	arrCylinderLink						: ARRAY [0..iMAX_CYLINDER_PAGES-1] OF ARRAY [0..iCYLINDERS_PER_PAGE-1] OF I_UniversalCylinder;				(*  *)
	arrAxisLink							: ARRAY [0..iMAX_AXIS_PAGES-1] OF ARRAY [0..iAXIS_PER_PAGE-1] OF I_UniversalAxis;							(*  *)
	arrInputLink						: ARRAY [0..iMAX_INPUT_PAGES-1] OF ARRAY [0..iINPUTS_PER_PAGE-1] OF I_DigitalInput;							(*  *)
	arrOutputLink						: ARRAY [0..iMAX_OUTPUT_PAGES-1] OF ARRAY [0..iOUTPUTS_PER_PAGE-1] OF I_DigitalOutput;						(*  *)
	arrSafeInputLink					: ARRAY	[0..iMAX_SAFE_INPUT_PAGES-1] OF ARRAY [0..iSAFE_INPUTS_PER_PAGE-1] OF I_DigitalInput;				(*  *)
	arrSafeOutputLink					: ARRAY [0..iMAX_SAFE_OUTPUT_PAGES-1] OF ARRAY [0..iSAFE_OUTPUTS_PER_PAGE-1] OF I_DigitalOutput;			(*  *)
	arrRobotLink						: ARRAY [0..iMAX_ROBOT_PAGES-1] OF ARRAY [0..iROBOTS_PER_PAGE-1] OF I_CR800EtherCAT;						(*  *)
	
	ifUniversalMachineLink				: I_UniversalMachine;	(*  *)
	ifRecipesManager					: I_RecipesManager;		(*  *)
	ifAlarmControler					: I_AlarmControler;		(*  *)
	
	(* --- Alarm page --- *)
	btnClearAll							: BOOL;	(*  *)
	btnExport							: BOOL;	(*  *)
	
	(* --- Recipes page --- *)
	(* Recipe control - buttons *)
	btnCreate							: BOOL;	(* Create recipe button *)
	btnSelect							: BOOL;	(* Select recipe from table button*)
	btnLoad								: BOOL;	(* Load recipe from file button *)
	btnRead								: BOOL;	(* Read recipe to file button *)
	btnReload 							: BOOL;	(* Reload recipes button *)
	btnBackup							: BOOL;	(* Backup recipes to external directory button *)
	btnRestore							: BOOL;	(* Restore recipes from external directory button *)
	btnRemove							: BOOL;	(* Remove recipe from the file *)
	btnReloadExternal					: BOOL;	(* Reload recipes button *)
	btnRecipeNext						: BOOL;	(* Go to next page with recipe parameters *)
	btnRecipePrevious					: BOOL;	(* Go to previous page with recipe parameters *)
	btnHmiClose							: BOOL;
	
	bUpdateVisuElements					: BOOL; (* For function block extending purposes (updating some visualisation elements after loading recipes) *)

	
	(* Recipe control - visibility *)
	bReloadInvisible					: BOOL;	(* Makes reload button invisible *)
	bRecipeNextInvisible				: BOOL;	(* Makes next button invisible *)
	bRecipePreviousInvisible			: BOOL;	(* Makes previous button invisible *)
	bRecipeCreateInvisible				: BOOL;	(* Makes create group box invisible *)
	bRecipeBackupRestoreInvisible		: BOOL;	(* Makes backup and restore group box invisible *)
	bNoRecipeSelected					: BOOL;
	
	(* Recipe control - control disabled *)
	bCreateRecipeDisabled				: BOOL;	(* Disable access to create recipe group box *)
	bBackupRestoreDisabled				: BOOL;	(* Disable access to backup and restore group box *)
	
	(* Recipe control - status *)
	bRecipesManagerError				: REFERENCE TO BOOL;					(* Error occured while executing last command *)
	eRecipesManagerReturns				: REFERENCE TO E_RecipesManagerReturns;	(* Result of last executed command *)
	
	(* Recipe control - parameters for recipes manager *)
	iSelectedRecipe						: INT;												(* Number of selected row in Available Recipes table *)
	sRecipeDefinition					: REFERENCE TO STRING;								(* Name of current recipe definition *)
	sSelectedRecipe						: STRING;											(* Current selected recipe name - changes affter trigger from btnSelect *)
	sNewRecipeName						: STRING;											(* Name for new recipe *)
	sBackupStoragePath					: STRING;											(* Path for backup/restoring of recipes *)
	arrRecipesNames						: REFERENCE TO ARRAY[0..127] OF STRING;				(* Names of all detected recipes *)
	sBackupRestoreRecipeName			: STRING;
		
	(* Recipe control - parameters frame generator *)
	iRecipeParameterIndex 				: USINT := 0;	(*  *)
	iRecipeParameterFrameIndex			: USINT := 0;	(*  *)	
	iRecipeParameterPageIndex			: USINT := 0;	(*  *)
	iSelectedRecipeParameterPageIndex	: USINT := 0;	(*  *)
	
	arrRecipeParameterFrameEmpty 		: ARRAY [0..iMAX_NUMBER_OF_RECIPES-1] OF ARRAY [0..iRECIPE_PARAMETERS_PER_PAGE-1] OF BOOL;							(*  *)
	arrRecipeParameterLink				: ARRAY [0..iMAX_NUMBER_OF_RECIPES-1] OF ARRAY [0..iRECIPE_PARAMETERS_PER_PAGE-1] OF I_RecipeParameter;				(*  *)
	arrRecipeParameterFrameData			: ARRAY [0..iMAX_NUMBER_OF_RECIPES-1] OF ARRAY [0..iRECIPE_PARAMETERS_PER_PAGE-1] OF ST_VisuCtrlRecipeParameter;	(*  *)
	arrRecipeParameterFrameType			: ARRAY [0..iMAX_NUMBER_OF_RECIPES-1] OF ARRAY [0..iRECIPE_PARAMETERS_PER_PAGE-1] OF E_VisuCtrlRecipeParameterType;	(*  *)
	
	(* --- Shell state machines --- *)
	eUniversalMachineCtrlState			: E_VisuCtrUniversalMachineState;		(*  *)
	eRecipesManagerState				: E_VisuCtrlRecipesManagerState;			(* Current state of Recipe Manager *)
	eAlarmCtrlState						: E_VisuCtrlAlarmControlState;			(* Current state of Alarm Controler *)
	
	(* --- Screen selectors --- *)
	eCurrentScreen						: E_VisuCtrlPageState;					(* Main page selector *)
	eLastScreen							: E_VisuCtrlPageState;					(* Last screen before change to auxilary screen *)
	eCurrentNavigation					: E_VisuCtrlNavBarState;				(* Navigation bar selector *)
	
	(* --- HMI buttons flags --- *)
	bStartDisable 						: BOOL;
	bStopDisable						: BOOL	:= TRUE;
	bVisNotInit 						: BOOL	:= TRUE;	
	bVisLogIn							: BOOL;
	bVisLogOut 							: BOOL	:= TRUE;	
	bVisHmiClose						: BOOL;
	bRecipeButtonDisabled				: BOOL;
	bModeSwitchButtonDisabled			: BOOL;
	                        			
	fbHmiClose							: NT_StartProcess;
END_VAR
(*
Version history:

+-------------+------------+----------------+----------+------------------------------------------+
|Date         | Version    | created under  | Author   | Remark                                   |
+=============+============+================+==========+==========================================+
|2022-03      | 1.0.0.0    | V3.1.4024.22   | ADBO     | Function block created                   |
+-------------+------------+----------------+----------+------------------------------------------+

*)

IF bFirstCycle THEN
	bFirstCycle := FALSE;
	(* Assign alarm references *)
	iActiveCriticals	REF= ifAlarmControler.ActiveCritical;
	iActvieErrors 		REF= ifAlarmControler.ActiveError;
	iActiveWarrnings	REF= ifAlarmControler.ActiveWarrning;
	
	(* Assign recipes references *)
	bRecipesManagerError 	REF= ifRecipesManager.Error;
	arrRecipesNames 		REF= ifRecipesManager.RecipesNames;
	eRecipesManagerReturns 	REF= ifRecipesManager.LastResult;
	sRecipeDefinition 		REF= ifRecipesManager.RecipesDefinition;
	
	(* --- Mark unused frames - saves CPU resources --- *)
	(* Cylinder frames *)
	FOR iLoop := 0 TO iMAX_CYLINDER_PAGES-1 DO
		FOR iLoop2 := 0 TO iCYLINDERS_PER_PAGE-1 DO
			IF arrCylinderLink[iLoop][iLoop2] = 0 THEN
				arrCylinderFrameEmpty[iLoop][iLoop2] := TRUE;
			END_IF
		END_FOR
	END_FOR
	
	(* Motor frames *)
	FOR iLoop := 0 TO iMAX_AXIS_PAGES-1 DO
		FOR iLoop2 := 0 TO iAXIS_PER_PAGE-1 DO
			IF arrAxisLink[iLoop][iLoop2] = 0 THEN
				arrAxisFrameEmpty[iLoop][iLoop2] := TRUE;
			END_IF
		END_FOR
	END_FOR
	
	(* Input frames *)
	FOR iLoop := 0 TO iMAX_INPUT_PAGES-1 DO
		FOR iLoop2 := 0 TO iINPUTS_PER_PAGE-1 DO
			IF arrInputLink[iLoop][iLoop2] = 0 THEN
				arrInputFrameEmpty[iLoop][iLoop2] := TRUE;
			END_IF
		END_FOR
	END_FOR
	
	(* Output frames *)
	FOR iLoop := 0 TO iMAX_OUTPUT_PAGES-1 DO
		FOR iLoop2 := 0 TO iOUTPUTS_PER_PAGE-1 DO
			IF arrOutputLink[iLoop][iLoop2] = 0 THEN
				arrOutputFrameEmpty[iLoop][iLoop2] := TRUE;
			END_IF
		END_FOR
	END_FOR
	
	(* Safe input frames *)
	FOR iLoop := 0 TO iMAX_SAFE_INPUT_PAGES-1 DO
		FOR iLoop2 := 0 TO iSAFE_INPUTS_PER_PAGE-1 DO
			IF arrSafeInputLink[iLoop][iLoop2] = 0 THEN
				arrSafeInputFrameEmpty[iLoop][iLoop2] := TRUE;
			END_IF
		END_FOR
	END_FOR
	
	(* Safe output frames *)
	FOR iLoop := 0 TO iMAX_SAFE_OUtPUT_PAGES-1 DO
		FOR iLoop2 := 0 TO iSAFE_OUtPUTS_PER_PAGE-1 DO
			IF arrSafeOutputLink[iLoop][iLoop2] = 0 THEN
				arrSafeOutputFrameEmpty[iLoop][iLoop2] := TRUE;
			END_IF
		END_FOR
	END_FOR
	
	(* Robot frames *)
	FOR iLoop := 0 TO iMAX_ROBOT_PAGES-1 DO
		FOR iLoop2 := 0 TO iROBOTS_PER_PAGE-1 DO
			IF arrRobotLink[iLoop][iLoop2] = 0 THEN
				arrRobotFrameEmpty[iLoop][iLoop2] := TRUE;
			END_IF
		END_FOR
	END_FOR
	
	(* Universal fixture frames *)
	//To-do
	
	(* Tcp-Server frames *)
	// To do
	
	(* Tcp-Client frames*)
	// To do
	
	(* Robot frames *)
	FOR iLoop := 0 TO iMAX_ROBOT_PAGES - 1 DO
		FOR iLoop2 := 0 TO iROBOTS_PER_PAGE - 1 DO
			IF arrRobotLink[iLoop][iLoop2] = 0 THEN
				arrRobotFrameEmpty[iLoop][iLoop2] := TRUE;
			END_IF
		END_FOR
	END_FOR
	
	(* Recipe parameters frames *)
	FOR iLoop := 0 TO iMAX_RECIPES_PAGES-1 DO
		FOR iLoop2 := 0 TO iRECIPE_PARAMETERS_PER_PAGE-1 DO
			IF arrRecipeParameterLink[iLoop][iLoop2] = 0 THEN
				arrRecipeParameterFrameEmpty[iLoop][iLoop2] := TRUE;
			END_IF
		END_FOR
	END_FOR
	
END_IF

(* Get current logged in user *)
IF btnLogIn AND LEN(WSTRING_TO_STRING(VisuUserManagement.VisuElems.CurrentFullUserName)) <> 0 THEN
	sCurrentUser := WSTRING_TO_STRING(VisuUserManagement.VisuElems.CurrentFullUserName);
	btnLogIn := FALSE;
ELSIF btnLogOut THEN
	MEMSET(ADR(sCurrentUser),0,SIZEOF(sCurrentUser));
	btnLogOut := FALSE;
END_IF

(* LogIn and LogOut button status flags *)
IF LEN(sCurrentUser) <> 0 THEN 
	bVisLogIn := TRUE;
	bVisLogOut:= FALSE;
	
ELSE
	bVisLogIn := FALSE;
	bVisLogOut:= TRUE;
	
END_IF

fbHmiClose(
	NETID			:= '',
	PATHSTR			:= 'C:\WINDOWS\system32\taskkill.exe' ,
	DIRNAME			:= '' ,
	COMNDLINE		:= '/t /f /IM Tc3PlcHmi.exe' , 
	START			:= btnHmiClose,
	ERRID			=> );

IF fbHmiClose.BUSY THEN		
	btnHmiClose := FALSE;	
END_IF

(* Get time and date *)
sCurrentDate := FUN_TimestructToDate(fbMachineTime.systemTime);
sCurrentTime := FUN_TimestructToTime(fbMachineTime.systemTime);
sCurrentTime := LEFT(STR := sCurrentTime, SIZE := (LEN(sCurrentTime)-4));

(* Universal switch to Alarms and Recipes page *)
IF btnRecipes THEN
	btnRecipes := FALSE;
	IF eCurrentScreen <> SCREEN_RECIPES AND eCurrentScreen <> SCREEN_ALARMS THEN
		eLastScreen := eCurrentScreen;
	END_IF
	eCurrentScreen := SCREEN_RECIPES;
	
ELSIF btnAlarms THEN
	btnAlarms := FALSE;
	IF eCurrentScreen <> SCREEN_RECIPES AND eCurrentScreen <> SCREEN_ALARMS THEN
		eLastScreen := eCurrentScreen;
	END_IF
	eCurrentScreen := SCREEN_ALARMS;
END_IF

(* Universal change to Abort - Reset mode *)
IF btnAbort THEN
	btnAbort := FALSE;
	eUniversalMachineCtrlState := VISU_CTRL_UNIVERSAL_MACHINE_ABORT;
	eAlarmCtrlState := VISU_CTRL_ALARM_CONTROLER_ABORT;
	eRecipesManagerState := VISU_CTRL_RECIPE_MANAGER_ABORT;
	eRecipesManagerState := VISU_CTRL_RECIPE_MANAGER_INIT;
	eCurrentScreen := SCREEN_ABORTING;
			
ELSIF btnReset THEN
	btnReset := FALSE;
	eUniversalMachineCtrlState := VISU_CTRL_UNIVERSAL_MACHINE_RESET;
END_IF

(* --- Alarm system control via shared interface --- *)
M_AlarmControler();

(* --- Recipes manager control via shared interface --- *)
M_RecipeManager();

(* --- Universal Machine control via shared interface ---*)
M_MachineControler();

(* --- Generic content control state machine --- *)
StateMachine();

PROPERTY Abort : REFERENCE TO BOOL
GET
Abort REF= btnAbort;
END_GET
END_PROPERTY

PROPERTY AutoMode : REFERENCE TO BOOL
GET
AutoMode REF= btnAuto;
END_GET
END_PROPERTY

PROPERTY Back : REFERENCE TO BOOL
GET
Back REF= btnBack;
END_GET
END_PROPERTY

PROPERTY Init : REFERENCE TO BOOL
GET
Init REF= btnInit;
END_GET
END_PROPERTY

METHOD PROTECTED M_AlarmControler
(* --- Active alarms counter --- *)
(*iActiveCriticals := ifAlarmControler.ActiveCritical;
iActvieErrors := ifAlarmControler.ActiveError;
iActiveWarrnings := ifAlarmControler.ActiveWarrning;*)
iActiveAlarms := iActvieErrors + iActiveCriticals;

(* Main alarm control via HMI *)
CASE eAlarmCtrlState OF
	VISU_CTRL_ALARM_CONTROLER_WAIT_FOR_CMD:
		IF btnInit THEN
			eAlarmCtrlState := VISU_CTRL_ALARM_CONTROLER_INIT;
			
		ELSIF btnClearAll THEN
			eAlarmCtrlState := VISU_CTRL_ALARM_CONTROLER_CLEAR_ALL; 
			
		ELSIF btnExport THEN
			eAlarmCtrlState := VISU_CTRL_ALARM_CONTTOLER_EXPORT;
			
		END_IF
		
	VISU_CTRL_ALARM_CONTROLER_INIT:
		ifAlarmControler.MR_Init();
		
		IF ifAlarmControler.Active THEN
			eAlarmCtrlState := VISU_CTRL_ALARM_CONTROLER_WAIT_FOR_CMD;
		END_IF
		
	VISU_CTRL_ALARM_CONTROLER_CLEAR_ALL:
		ifAlarmControler.MR_ClearAll(bResetConfirmation := TRUE);
		
		IF NOT ifAlarmControler.Busy THEN
			eAlarmCtrlState := VISU_CTRL_ALARM_CONTROLER_WAIT_FOR_CMD;
		END_IF
	
	VISU_CTRL_ALARM_CONTTOLER_EXPORT:
		ifAlarmControler.MR_Export();
		
		IF NOT ifAlarmControler.Busy THEN
			eAlarmCtrlState := VISU_CTRL_ALARM_CONTROLER_WAIT_FOR_CMD;
		END_IF
		
	VISU_CTRL_ALARM_CONTROLER_ABORT:
		ifAlarmControler.MR_Abort();
		
		IF NOT ifAlarmControler.Active THEN
			eAlarmCtrlState := VISU_CTRL_ALARM_CONTROLER_WAIT_FOR_CMD;
		END_IF
		
END_CASE
END_METHOD

METHOD M_MachineControler : BOOL
(* Main machine control via HMI *)
IF NOT ifUniversalMachineLink.Running THEN
	bStartDisable := FALSE;
	bStopDisable := TRUE;
ELSE
	bStartDisable := TRUE;
	bStopDisable := FALSE;
END_IF

CASE eUniversalMachineCtrlState OF
	VISU_CTRL_UNIVERSAL_MACHINE_WAIT_FOR_CMD:
		IF btnInit THEN
			eUniversalMachineCtrlState := VISU_CTRL_UNIVERSAL_MACHINE_INIT;
			
		ELSIF btnStart THEN
			eUniversalMachineCtrlState := VISU_CTRL_UNIVERSAL_MACHINE_START_AUTO;
			
		ELSIF btnStop THEN
			eUniversalMachineCtrlState := VISU_CTRL_UNIVERSAL_MACHINE_STOP_AUTO;
			
		ELSIF btnManual THEN
			eUniversalMachineCtrlState := VISU_CTRL_UNIVERSAL_MACHINE_SWITCH_TO_MANUAL;
			
		ELSIF btnAuto THEN
			eUniversalMachineCtrlState := VISU_CTRL_UNIVERSAL_MACHINE_SWITCH_TO_AUTO;
			
		ELSIF btnAbort THEN
			eUniversalMachineCtrlState := VISU_CTRL_UNIVERSAL_MACHINE_ABORT;
			
		ELSIF btnReset THEN
			eUniversalMachineCtrlState := VISU_CTRL_UNIVERSAL_MACHINE_RESET;			
		END_IF
	
	VISU_CTRL_UNIVERSAL_MACHINE_INIT:
		ifUniversalMachineLink.MR_Init();
		
		IF ifUniversalMachineLink.Active THEN
			bVisNotInit := FALSE;
			bVisHmiClose:= TRUE;
						
			eUniversalMachineCtrlState := VISU_CTRL_UNIVERSAL_MACHINE_WAIT_FOR_CMD;
		END_IF
	
	VISU_CTRL_UNIVERSAL_MACHINE_RESET:
		ifUniversalMachineLink.MR_Reset();
		
		IF NOT ifUniversalMachineLink.Error THEN
			eUniversalMachineCtrlState := VISU_CTRL_UNIVERSAL_MACHINE_WAIT_FOR_CMD;
		END_IF
	
	VISU_CTRL_UNIVERSAL_MACHINE_START_AUTO:
		ifUniversalMachineLink.MR_Start();
		
		IF ifUniversalMachineLink.Running THEN
			eUniversalMachineCtrlState := VISU_CTRL_UNIVERSAL_MACHINE_WAIT_FOR_CMD;
		END_IF
	
	VISU_CTRL_UNIVERSAL_MACHINE_STOP_AUTO:
		ifUniversalMachineLink.MR_Stop();
		
		IF NOT ifUniversalMachineLink.Running THEN
			eUniversalMachineCtrlState := VISU_CTRL_UNIVERSAL_MACHINE_WAIT_FOR_CMD;
		END_IF
		
	VISU_CTRL_UNIVERSAL_MACHINE_SWITCH_TO_MANUAL:
		ifUniversalMachineLink.MR_SwitchToManual();
		
		IF ifUniversalMachineLink.State = MACHINE_STATE_MANUAL THEN
			eUniversalMachineCtrlState := VISU_CTRL_UNIVERSAL_MACHINE_WAIT_FOR_CMD;
		END_IF
	
	VISU_CTRL_UNIVERSAL_MACHINE_SWITCH_TO_AUTO:
		ifUniversalMachineLink.MR_SwitchToAuto();
		
		IF ifUniversalMachineLink.State = MACHINE_STATE_AUTO THEN
			eUniversalMachineCtrlState := VISU_CTRL_UNIVERSAL_MACHINE_WAIT_FOR_CMD;
		END_IF
	
	VISU_CTRL_UNIVERSAL_MACHINE_ABORT:
		ifUniversalMachineLink.MR_Abort();
		
		IF NOT ifUniversalMachineLink.Active THEN
			bVisNotInit := TRUE;
			bVisHmiClose:= FALSE;
			
			eUniversalMachineCtrlState := VISU_CTRL_UNIVERSAL_MACHINE_WAIT_FOR_CMD;
		END_IF
		
END_CASE
END_METHOD

METHOD PROTECTED M_RecipeManager
bRecipesManagerError 	:= ifRecipesManager.Error;
arrRecipesNames 		:= ifRecipesManager.RecipesNames;
eRecipesManagerReturns 	:= ifRecipesManager.LastResult;
sRecipeDefinition 		:= ifRecipesManager.RecipesDefinition;

IF bStartDisable OR bVisNotInit THEN
	bRecipeButtonDisabled := TRUE;
ELSE
	bRecipeButtonDisabled := FALSE;
END_IF

(* Previous page button visiblity control *)
IF iSelectedRecipeParameterPageIndex = 0 THEN
	bRecipePreviousInvisible := TRUE;
ELSE
	bRecipePreviousInvisible := FALSE;
END_IF

IF sSelectedRecipe = '' THEN
	bNoRecipeSelected := TRUE;

ELSE 
	bNoRecipeSelected := FALSE;

END_IF

(* Next page button visibility control *)
IF btnRecipeNext THEN
	btnRecipeNext := FALSE;
	iSelectedRecipeParameterPageIndex := iSelectedRecipeParameterPageIndex + 1;
	
ELSIF btnRecipePrevious THEN
	btnRecipePrevious := FALSE;
	iSelectedRecipeParameterPageIndex := iSelectedRecipeParameterPageIndex - 1;
END_IF

(* Selecting new recipe from table *)
IF btnSelect THEN
	btnSelect := FALSE;
	sSelectedRecipe	:= arrRecipesNames[iSelectedRecipe];
	eRecipesManagerState := VISU_CTRL_RECIPE_MANAGER_RELOAD;
END_IF

(* Main recipe manager control via HMI *)
CASE eRecipesManagerState OF
	VISU_CTRL_RECIPE_MANAGER_WAIT_FOR_CMD:
		IF btnInit THEN
			eRecipesManagerState := VISU_CTRL_RECIPE_MANAGER_INIT;
			
		ELSIF btnCreate THEN
			btnCreate := FALSE;
			eRecipesManagerState := VISU_CTRL_RECIPE_MANAGER_CREATE;
			
		ELSIF btnLoad THEN
			btnLoad := FALSE;
			eRecipesManagerState := VISU_CTRL_RECIPE_MANAGER_LOAD;
			
		ELSIF btnRead THEN
			btnRead := FALSE;
			eRecipesManagerState := VISU_CTRL_RECIPE_MANAGER_READ;
			
		ELSIF btnReload THEN
			btnReload := FALSE;
			eRecipesManagerState := VISU_CTRL_RECIPE_MANAGER_RELOAD;	
						
		ELSIF btnReloadExternal THEN
			btnReloadExternal := FALSE;
			eRecipesManagerState := VISU_CTRL_RECIPE_MANAGER_RELOAD_EXT;
			
		ELSIF btnBackup THEN
			btnBackup := FALSE;
			eRecipesManagerState := VISU_CTRL_RECIPE_MANAGER_BACKUP;
			
		ELSIF btnRestore THEN
			btnRestore := FALSE;
			eRecipesManagerState := VISU_CTRL_RECIPE_MANAGER_RESTORE;
			
		ELSIF btnRemove THEN
			btnRemove := FALSE;
			eRecipesManagerState := VISU_CTRL_RECIPE_MANAGER_REMOVE;
						
		END_IF
		
	VISU_CTRL_RECIPE_MANAGER_INIT:
		ifRecipesManager.MR_Init();
		
		IF ifRecipesManager.Active THEN
			eRecipesManagerState := VISU_CTRL_RECIPE_MANAGER_WAIT_FOR_CMD;
		END_IF
	
	VISU_CTRL_RECIPE_MANAGER_CREATE:
		ifRecipesManager.MR_Create( sRecipesDefinition	:= sRecipeDefinition,
									sRecipeName			:= sNewRecipeName);
									
		IF NOT ifRecipesManager.Busy THEN
			eRecipesManagerState := VISU_CTRL_RECIPE_MANAGER_WAIT_FOR_CMD;
		END_IF
	
	VISU_CTRL_RECIPE_MANAGER_LOAD:
		ifRecipesManager.MR_LoadAndWritte( 	sRecipesDefinition	:= sRecipeDefinition,
											sRecipeName			:= sSelectedRecipe);
									
		IF NOT ifRecipesManager.Busy THEN
			IF NOT ifRecipesManager.Error THEN
				sCurrentRecipe := sSelectedRecipe; 
			END_IF
			
			bUpdateVisuElements := TRUE;
			eRecipesManagerState := VISU_CTRL_RECIPE_MANAGER_WAIT_FOR_CMD;
		END_IF
	
	VISU_CTRL_RECIPE_MANAGER_READ:
		ifRecipesManager.MR_ReadAndSave(	sRecipesDefinition	:= sRecipeDefinition,
											sRecipeName			:= sSelectedRecipe);
									
		IF NOT ifRecipesManager.Busy THEN
			eRecipesManagerState := VISU_CTRL_RECIPE_MANAGER_WAIT_FOR_CMD;
		END_IF
	
	VISU_CTRL_RECIPE_MANAGER_RELOAD:
		ifRecipesManager.MR_Reload( sRecipesDefinition := sRecipeDefinition,
									sRecipeName := sSelectedRecipe);
									
		IF NOT ifRecipesManager.Busy THEN
			eRecipesManagerState := VISU_CTRL_RECIPE_MANAGER_WAIT_FOR_CMD;
		END_IF
		
	VISU_CTRL_RECIPE_MANAGER_RELOAD_EXT:
		ifRecipesManager.MR_ReloadExternal( sRecipesDefinition := sRecipeDefinition,
											sRecipeName := sBackupRestoreRecipeName,
											sBackupStoragePath := sBackupStoragePath);
									
		IF NOT ifRecipesManager.Busy THEN
			eRecipesManagerState := VISU_CTRL_RECIPE_MANAGER_WAIT_FOR_CMD;
		END_IF	
	
	VISU_CTRL_RECIPE_MANAGER_BACKUP:
		ifRecipesManager.MR_Backup(sRecipesDefinition := sRecipeDefinition,
									sRecipeName := sBackupRestoreRecipeName,
									sBackupStoragePath := sBackupStoragePath);
									
		IF NOT ifRecipesManager.Busy THEN
			eRecipesManagerState := VISU_CTRL_RECIPE_MANAGER_WAIT_FOR_CMD;
		END_IF
		
	VISU_CTRL_RECIPE_MANAGER_RESTORE:
		ifRecipesManager.MR_Restore(sRecipesDefinition := sRecipeDefinition,
									sRecipeName := sBackupRestoreRecipeName,
									sBackupStoragePath := sBackupStoragePath);
									
		IF NOT ifRecipesManager.Busy THEN
			IF NOT ifRecipesManager.Error THEN
				sCurrentRecipe := sSelectedRecipe; 
			END_IF
			
			bUpdateVisuElements := TRUE;
			eRecipesManagerState := VISU_CTRL_RECIPE_MANAGER_WAIT_FOR_CMD;
		END_IF
		
	VISU_CTRL_RECIPE_MANAGER_REMOVE:
		ifRecipesManager.MR_Remove( sRecipesDefinition := sRecipeDefinition,
									sRecipeName := sSelectedRecipe);
		
		IF NOT ifRecipesManager.Busy THEN
			eRecipesManagerState := VISU_CTRL_RECIPE_MANAGER_WAIT_FOR_CMD;
		END_IF
	
	VISU_CTRL_RECIPE_MANAGER_ABORT:
		ifRecipesManager.MR_Abort();
		
		IF NOT ifRecipesManager.Active THEN
			eRecipesManagerState := VISU_CTRL_RECIPE_MANAGER_WAIT_FOR_CMD;
		END_IF
	
END_CASE
END_METHOD

PROPERTY ManualMode : REFERENCE TO BOOL
GET
ManualMode REF= btnManual;
END_GET
END_PROPERTY

METHOD MR_AppendAlarmControler : BOOL
VAR_INPUT
	ifAlarmControler : I_AlarmControler;
END_VAR
THIS^.ifAlarmControler := ifAlarmControler;
MR_AppendAlarmControler := TRUE;
END_METHOD

METHOD MR_AppendAxis : BOOL
VAR_INPUT
	ifMotor 	: I_UniversalAxis;
	eMotorType	: E_VisuCtrlAxisImgType;
END_VAR
IF iAxisIndex < iMAX_AXIS_FRAMES THEN
	arrAxisLink[iAxisPageIndex][iAxisFrameIndex] := ifMotor;
	arrAxisFrameEmpty[iAxisPageIndex][iAxisFrameIndex] := FALSE;
	arrAxisFrame[iAxisPageIndex][iAxisFrameIndex].sAxisImage := TO_STRING(eMotorType);
	
	IF iAxisFrameIndex = iAXIS_PER_PAGE - 1 THEN
		iAxisPageIndex := iAxisPageIndex + 1;
		iAxisFrameIndex := 0;
	ELSE
		iAxisFrameIndex := iAxisFrameIndex + 1;
	END_IF	

	iAxisIndex := iAxisIndex + 1;
	MR_AppendAxis := TRUE;
ELSE
	MR_AppendAxis := FALSE;
END_IF
END_METHOD

METHOD MR_AppendCylinder : BOOL
VAR_INPUT
	ifCylinder			: I_UniversalCylinder;
	eCylinderType		: E_VisuCtrlCylinderImgType;
	sActiveDescription	: STRING;
	sHomeDescription	: STRING;
END_VAR
IF iCylinderIndex < iMAX_CYLINDER_FRAMES THEN
	arrCylinderLink[iCylinderPageIndex][iCylinderFrameIndex] := ifCylinder;
	arrCylinderFrameEmpty[iCylinderPageIndex][iCylinderFrameIndex] := FALSE;
	
	arrCylinderFrame[iCylinderPageIndex][iCylinderFrameIndex].sCylinderImage := TO_STRING(eCylinderType);
	arrCylinderFrame[iCylinderPageIndex][iCylinderFrameIndex].sActiveDescription := sActiveDescription;
	arrCylinderFrame[iCylinderPageIndex][iCylinderFrameIndex].sHomeDescription := sHomeDescription;
	
	IF iCylinderFrameIndex = iCYLINDERS_PER_PAGE - 1 THEN
		iCylinderPageIndex := iCylinderPageIndex + 1;
		iCylinderFrameIndex := 0;
	ELSE
		iCylinderFrameIndex := iCylinderFrameIndex + 1;
	END_IF	

	iCylinderIndex := iCylinderIndex + 1;
	MR_AppendCylinder := TRUE;
ELSE
	MR_AppendCylinder := FALSE;
END_IF
END_METHOD

METHOD MR_AppendInput : BOOL
VAR_INPUT
	ifDigitalInput : I_DigitalInput;
END_VAR
IF iInputIndex < iMAX_INPUT_FRAMES THEN
	arrInputLink[iInputPageIndex][iInputFrameIndex] := ifDigitalInput;
	arrInputFrameEmpty[iInputPageIndex][iInputFrameIndex] := FALSE;
	
	IF iInputFrameIndex = iINPUTS_PER_PAGE - 1 THEN
		iInputPageIndex := iInputPageIndex + 1;
		iInputFrameIndex := 0;
	ELSE
		iInputFrameIndex := iInputFrameIndex + 1;
	END_IF	
	
	iInputIndex := iInputIndex + 1;
	MR_AppendInput := TRUE;
ELSE
	MR_AppendInput := FALSE;
END_IF
END_METHOD

METHOD MR_AppendOutput : BOOL
VAR_INPUT
	ifDigitalOutput : I_DigitalOutput;
END_VAR
IF iOutputIndex < iMAX_OUTPUT_FRAMES THEN
	arrOutputLink[iOutputPageIndex][iOutputFrameIndex] := ifDigitalOutput;
	arrOutputFrameEmpty[iOutputPageIndex][iOutputFrameIndex] := FALSE;
	
	IF iOutputFrameIndex = iOUTPUTS_PER_PAGE - 1 THEN
		iOutputPageIndex := iOutputPageIndex + 1;
		iOutputFrameIndex := 0;
	ELSE
		iOutputFrameIndex := iOutputFrameIndex + 1;
	END_IF	

	iOutputIndex := iOutputIndex + 1;
	MR_AppendOutput := TRUE;
ELSE
	MR_AppendOutput := FALSE;
END_IF
END_METHOD

METHOD MR_AppendRecipeParameter : BOOL
VAR_INPUT
	ifRecipeParameter : I_RecipeParameter;
END_VAR
IF iRecipeParameterIndex < iMAX_NUMBER_OF_RECIPES THEN
	arrRecipeParameterLink[iRecipeParameterPageIndex][iRecipeParameterFrameIndex] 		:= ifRecipeParameter;
	arrRecipeParameterFrameEmpty[iRecipeParameterPageIndex][iRecipeParameterFrameIndex] := FALSE;
	arrRecipeParameterFrameType[iRecipeParameterPageIndex][iRecipeParameterFrameIndex]	:= ifRecipeParameter.DataType;
	
	arrRecipeParameterFrameData[iRecipeParameterPageIndex][iRecipeParameterFrameIndex].bValue 		REF= arrRecipeParameterLink[iRecipeParameterPageIndex][iRecipeParameterFrameIndex].BitValue;
	arrRecipeParameterFrameData[iRecipeParameterPageIndex][iRecipeParameterFrameIndex].iValue 		REF= arrRecipeParameterLink[iRecipeParameterPageIndex][iRecipeParameterFrameIndex].IntValue;
	arrRecipeParameterFrameData[iRecipeParameterPageIndex][iRecipeParameterFrameIndex].rValue 		REF= arrRecipeParameterLink[iRecipeParameterPageIndex][iRecipeParameterFrameIndex].RealValue;
	arrRecipeParameterFrameData[iRecipeParameterPageIndex][iRecipeParameterFrameIndex].sValue 		REF= arrRecipeParameterLink[iRecipeParameterPageIndex][iRecipeParameterFrameIndex].StringValue;
	arrRecipeParameterFrameData[iRecipeParameterPageIndex][iRecipeParameterFrameIndex].sName 		REF= arrRecipeParameterLink[iRecipeParameterPageIndex][iRecipeParameterFrameIndex].Name;
	arrRecipeParameterFrameData[iRecipeParameterPageIndex][iRecipeParameterFrameIndex].sFileValue 	REF= arrRecipeParameterLink[iRecipeParameterPageIndex][iRecipeParameterFrameIndex].FileValue;
	
	IF iRecipeParameterFrameIndex = iRECIPE_PARAMETERS_PER_PAGE - 1 THEN
		iRecipeParameterPageIndex := iRecipeParameterPageIndex + 1;
		iRecipeParameterFrameIndex := 0;
	ELSE
		iRecipeParameterFrameIndex := iRecipeParameterFrameIndex + 1;
	END_IF	
	
	iRecipeParameterIndex := iRecipeParameterIndex + 1;
	MR_AppendRecipeParameter := FALSE;
ELSE
	MR_AppendRecipeParameter := FALSE;
END_IF
END_METHOD

METHOD MR_AppendRecipesManager : BOOL
VAR_INPUT
	ifRecipesManager : I_RecipesManager;
END_VAR
THIS^.ifRecipesManager := ifRecipesManager;
MR_AppendRecipesManager := TRUE;
END_METHOD

METHOD MR_AppendRobot : BOOL
VAR_INPUT
	ifRobot				: I_CR800EtherCAT;
	eRobotType			: E_VisuCtrlRobotImgType;
//	sErrorDescription	: STRING;
END_VAR
IF iRobotIndex < iMAX_ROBOT_FRAMES THEN
	arrRobotLink[iRobotPageIndex][iRobotFrameIndex] := ifRobot;
	arrRobotFrameEmpty[iRobotPageIndex][iRobotFrameIndex] := FALSE;
	arrRobotFrame[iRobotPageIndex][iRobotFrameIndex].sRobotImage := TO_STRING(eRobotType);
	
	IF iRobotFrameIndex = iROBOTS_PER_PAGE - 1 THEN
		iRobotPageIndex := iRobotPageIndex + 1;
		iRobotFrameIndex := 0;
	ELSE
		iRobotFrameIndex := iRobotFrameIndex + 1;
	END_IF	

	iRobotIndex := iRobotIndex + 1;
	MR_AppendRobot := TRUE;
ELSE
	MR_AppendRobot := FALSE;
END_IF
END_METHOD

METHOD MR_AppendSafeInput : BOOL
VAR_INPUT
	ifSafeInput : I_DigitalInput;
END_VAR
IF iSafeInputIndex < iMAX_SAFE_INPUT_FRAMES THEN
	arrSafeInputLink[iSafeInputPageIndex][iSafeInputFrameIndex] := ifSafeInput;
	arrSafeInputFrameEmpty[iSafeInputPageIndex][iSafeInputFrameIndex] := FALSE;
	
	IF iSafeInputFrameIndex = iSAFE_INPUTS_PER_PAGE - 1 THEN
		iSafeInputPageIndex := iSafeInputPageIndex + 1;
		iSafeInputFrameIndex := 0;
	ELSE
		iSafeInputFrameIndex := iSafeInputFrameIndex + 1;
	END_IF	
	
	iSafeInputIndex := iSafeInputIndex + 1;
	MR_AppendSafeInput := TRUE;
ELSE
	MR_AppendSafeInput := FALSE;
END_IF
END_METHOD

METHOD MR_AppendSafeOutput : BOOL
VAR_INPUT
	ifSafeOutput : I_DigitalOutput;
END_VAR
IF iSafeOutputIndex < iMAX_SAFE_OUTPUT_FRAMES THEN
	arrSafeOutputLink[iSafeOutputPageIndex][iSafeOutputFrameIndex] := ifSafeOutput;
	arrSafeOutputFrameEmpty[iSafeOutputPageIndex][iSafeOutputFrameIndex] := FALSE;
	
	IF iSafeOutputFrameIndex = iSAFE_OUTPUTS_PER_PAGE - 1 THEN
		iSafeOutputPageIndex := iSafeOutputPageIndex + 1;
		iSafeOutputFrameIndex := 0;
	ELSE
		iSafeOutputFrameIndex := iSafeOutputFrameIndex + 1;
	END_IF		

	iSafeOutputIndex := iSafeOutputIndex + 1;
	MR_AppendSafeOutput := TRUE;
ELSE
	MR_AppendSafeOutput := FALSE;
END_IF
END_METHOD

METHOD MR_AppendUniversalMachine : BOOL
VAR_INPUT
	ifMachine : I_UniversalMachine;
END_VAR
THIS^.ifUniversalMachineLink := ifMachine;
MR_AppendUniversalMachine := TRUE;
END_METHOD

METHOD MR_FirstCycle : BOOL
VAR_INPUT
	sMachineName : STRING;
	sSoftwareVersion : STRING;
END_VAR
THIS^.sMachineName := sMachineName;
THIS^.sSoftwareVersion := sSoftwareVersion;
END_METHOD

METHOD PROTECTED MS_Aborting
VAR_INPUT
END_VAR
eCurrentNavigation := NAVIGATION_EMPTY;

IF ifUniversalMachineLink.State = MACHINE_STATE_UNINITIALIZED THEN
	eCurrentScreen := SCREEN_UNINITIALIZED;
	
ELSIF ifUniversalMachineLink.State = MACHINE_STATE_EMERGENCY THEN
	eCurrentScreen := SCREEN_EMERGENCY;
	
END_IF
END_METHOD

METHOD PROTECTED MS_Alarms
VAR_INPUT
END_VAR
eCurrentNavigation := NAVIGATION_UTILITIES;

IF btnBack THEN
	btnBack := FALSE;
	eCurrentScreen := eLastScreen;
END_IF
END_METHOD

METHOD PROTECTED MS_Auto
VAR_INPUT
END_VAR
eCurrentNavigation := NAVIGATION_AUTO;

IF ifUniversalMachineLink.State = MACHINE_STATE_ABORTING THEN
	eCurrentScreen := SCREEN_ABORTING;	

ELSIF ifUniversalMachineLink.State = MACHINE_STATE_AUTO_TO_MANUAL THEN
	eCurrentScreen := SCREEN_MODE_CHANGE;
	
	IF iOutputIndex > 0 THEN
		FOR iLoop := 0 TO iOUTPUTS_PER_PAGE-1 DO
			IF arrOutputFrameEmpty[iSelectedOutputPageIndex][iLoop] = FALSE THEN
				arrOutputFrame[iSelectedOutputPageIndex][iLoop].btnOut := arrOutputLink[iSelectedOutputPageIndex][iLoop].Out;
				
				IF arrOutputFrameEmpty[iSelectedOutputPageIndex][iLoop +1 ] = TRUE THEN
					EXIT;
					
				END_IF
			END_IF
		END_FOR
	END_IF
ELSIF ifUniversalMachineLink.State = MACHINE_STATE_EMERGENCY THEN
	eCurrentScreen := SCREEN_EMERGENCY;
	
END_IF
END_METHOD

METHOD PROTECTED ABSTRACT MS_Emergency
END_METHOD

METHOD PROTECTED MS_Initializing
VAR_INPUT
END_VAR
eCurrentNavigation := NAVIGATION_INITIALIZING;

IF ifUniversalMachineLink.State = MACHINE_STATE_UNINITIALIZED THEN
	eCurrentScreen := SCREEN_UNINITIALIZED;
			
ELSIF ifUniversalMachineLink.State = MACHINE_STATE_READY_INITIALIZED THEN
	eCurrentScreen := SCREEN_READY_INITIALIZED;
	
ELSIF ifUniversalMachineLink.State = MACHINE_STATE_AUTO THEN
	eCurrentScreen := SCREEN_AUTO;
	
ELSIF ifUniversalMachineLink.State = MACHINE_STATE_EMERGENCY THEN
	eCurrentScreen := SCREEN_EMERGENCY;
			
END_IF
END_METHOD

METHOD PROTECTED MS_Manual
VAR_INPUT
END_VAR
eCurrentNavigation := NAVIGATION_MANUAL;

IF ifUniversalMachineLink.State = MACHINE_STATE_UNINITIALIZED THEN
	eCurrentScreen := SCREEN_UNINITIALIZED;	
	
ELSIF ifUniversalMachineLink.State = MACHINE_STATE_MANUAL_TO_AUTO THEN
	eCurrentScreen := SCREEN_MODE_CHANGE;
	
ELSIF ifUniversalMachineLink.State = MACHINE_STATE_EMERGENCY THEN
	eCurrentScreen := SCREEN_EMERGENCY;
	
END_IF

IF btnManualCylinder THEN
	eCurrentScreen := SCREEN_MANUAL_CYLINDERS;

ELSIF btnManualAxis THEN
	eCurrentScreen := SCREEN_MANUAL_MOTORS;
	
ELSIF btnManualInputs THEN
	eCurrentScreen := SCREEN_MANUAL_INPUTS;
	
ELSIF btnManualOutputs THEN
	eCurrentScreen := SCREEN_MANUAL_OUTPUTS;
	
//ELSIF btnManualSafety THEN
//	eCurrentScreen := SCREEN_MANUAL_SAFETY;

ELSIF btnManualRobots THEN
	eCurrentScreen := SCREEN_MANUAL_ROBOTS;

ELSIF btnManualOthers THEN
	eCurrentScreen := SCREEN_MANUAL_OTHERS;
	
END_IF
END_METHOD

METHOD PROTECTED MS_ManualAxis
VAR_INPUT
END_VAR
(*Set current screen *)
eCurrentScreen := SCREEN_MANUAL_MOTORS;

(* Run common part of manual pages handling *)
MS_Manual();

IF arrAxisFrameEmpty[iAxisPageIndex][0] THEN
    iAxisPageIndex := iAxisPageIndex - 1;
END_IF

bNextInvisible := iSelectedAxisPageIndex = iAxisPageIndex;
bPreviousInvisible := iSelectedAxisPageIndex = 0;

(* Frames control *)
IF btnPrevious THEN
	btnPrevious := FALSE;
	iSelectedAxisPageIndex := iSelectedAxisPageIndex - 1;
ELSIF btnNext THEN
	btnNext := FALSE;
	iSelectedAxisPageIndex := iSelectedAxisPageIndex + 1;
END_IF

IF iAxisIndex > 0 THEN
	FOR iLoop := 0 TO iAXIS_PER_PAGE-1 DO
		IF arrAxisFrameEmpty[iSelectedAxisPageIndex][iLoop] = FALSE THEN
			(* Assign object status to frame*)
			arrAxisFrame[iSelectedAxisPageIndex][iLoop].bActive := arrAxisLink[iSelectedAxisPageIndex][iLoop].Active;
			arrAxisFrame[iSelectedAxisPageIndex][iLoop].bHomed := arrAxisLink[iSelectedAxisPageIndex][iLoop].IsHomed;
			arrAxisFrame[iSelectedAxisPageIndex][iLoop].bInPosition := arrAxisLink[iSelectedAxisPageIndex][iLoop].InPosition;
			arrAxisFrame[iSelectedAxisPageIndex][iLoop].bHalted := arrAxisLink[iSelectedAxisPageIndex][iLoop].Halted;
			arrAxisFrame[iSelectedAxisPageIndex][iLoop].bError := arrAxisLink[iSelectedAxisPageIndex][iLoop].Error;
			arrAxisFrame[iSelectedAxisPageIndex][iLoop].iErrorID := arrAxisLink[iSelectedAxisPageIndex][iLoop].ErrorID;
			arrAxisFrame[iSelectedAxisPageIndex][iLoop].eAxisState := arrAxisLink[iSelectedAxisPageIndex][iLoop].State;
			arrAxisFrame[iSelectedAxisPageIndex][iLoop].lrActualPosition := arrAxisLink[iSelectedAxisPageIndex][iLoop].ActualPosition;
			arrAxisFrame[iSelectedAxisPageIndex][iLoop].lrActualVelocity := arrAxisLink[iSelectedAxisPageIndex][iLoop].ActualVelocity;
			arrAxisFrame[iSelectedAxisPageIndex][iLoop].lrSetPosition := arrAxisLink[iSelectedAxisPageIndex][iLoop].SetpointPosition;
			arrAxisFrame[iSelectedAxisPageIndex][iLoop].lrSetVelocity := arrAxisLink[iSelectedAxisPageIndex][iLoop].SetpointVelocity;
			arrAxisFrame[iSelectedAxisPageIndex][iLoop].lrLagError := arrAxisLink[iSelectedAxisPageIndex][iLoop].LagError;
			arrAxisFrame[iSelectedAxisPageIndex][iLoop].sName := arrAxisLink[iSelectedAxisPageIndex][iLoop].Name;
			arrAxisFrame[iSelectedAxisPageIndex][iLoop].sUnit := arrAxisLink[iSelectedAxisPageIndex][iLoop].Unit;
			
			(* Assign parameters from frame to object *)
			arrAxisLink[iSelectedAxisPageIndex][iLoop].Override := arrAxisFrame[iSelectedAxisPageIndex][iLoop].lrOverride;
			arrAxisLink[iSelectedAxisPageIndex][iLoop].JogPosition := arrAxisFrame[iSelectedAxisPageIndex][iLoop].lrJogDistance;
			arrAxisLink[iSelectedAxisPageIndex][iLoop].JogVelocity := arrAxisFrame[iSelectedAxisPageIndex][iLoop].lrJogVelocity;
			arrAxisLink[iSelectedAxisPageIndex][iLoop].JogAcceleration := arrAxisFrame[iSelectedAxisPageIndex][iLoop].lrJogAcceleration;
			arrAxisLink[iSelectedAxisPageIndex][iLoop].JogDeceleration := arrAxisFrame[iSelectedAxisPageIndex][iLoop].lrJogDeceleartion;
			
			(* Bound jog mode frame selector to axis object jog mode *)
			CASE arrAxisFrame[iSelectedAxisPageIndex][iLoop].eJogMode OF
				VISU_AXIS_JOG_MODE_STANDARD_SLOW:
					arrAxisLink[iSelectedAxisPageIndex][iLoop].JogMode := E_JogMode.MC_JOGMODE_STANDARD_SLOW;
					
				VISU_AXIS_JOG_MODE_STANDARD_FAST:
					arrAxisLink[iSelectedAxisPageIndex][iLoop].JogMode := E_JogMode.MC_JOGMODE_STANDARD_FAST;
					
				VISU_AXIS_JOG_MODE_CONTINOUS:
					arrAxisLink[iSelectedAxisPageIndex][iLoop].JogMode := E_JogMode.MC_JOGMODE_CONTINOUS;
					
				VISU_AXIS_JOG_MODE_INCHING:
					arrAxisLink[iSelectedAxisPageIndex][iLoop].JogMode := E_JogMode.MC_JOGMODE_INCHING;
					
				VISU_AXIS_JOG_MODE_INCHING_MODULO:
					arrAxisLink[iSelectedAxisPageIndex][iLoop].JogMode := E_JogMode.MC_JOGMODE_INCHING_MODULO;
					
			END_CASE
			
			(* Manual object control via requests *)
			IF arrAxisFrame[iSelectedAxisPageIndex][iLoop].btnReset THEN
				arrAxisFrame[iSelectedAxisPageIndex][iLoop].btnReset := FALSE;
				arrAxisState[iSelectedAxisPageIndex][iLoop] := VISU_CTRL_AXIS_RESET;
				
			ELSIF arrAxisFrame[iSelectedAxisPageIndex][iLoop].btnHalt THEN
				arrAxisFrame[iSelectedAxisPageIndex][iLoop].btnHalt := FALSE;
				arrAxisState[iSelectedAxisPageIndex][iLoop] := VISU_CTRL_AXIS_HALT;
				
			END_IF
			
			CASE arrAxisState[iSelectedAxisPageIndex][iLoop] OF
				VISU_CTRL_AXIS_WAIT_FOR_CMD:
					IF arrAxisFrame[iSelectedAxisPageIndex][iLoop].btnInit THEN
						arrAxisFrame[iSelectedAxisPageIndex][iLoop].btnInit := FALSE;
						arrAxisState[iSelectedAxisPageIndex][iLoop] := VISU_CTRL_AXIS_INIT;
						
					ELSIF arrAxisFrame[iSelectedAxisPageIndex][iLoop].btnHome THEN
						arrAxisFrame[iSelectedAxisPageIndex][iLoop].btnHome := FALSE;
						arrAxisState[iSelectedAxisPageIndex][iLoop] := VISU_CTRL_AXIS_HOME;
						
					ELSIF arrAxisFrame[iSelectedAxisPageIndex][iLoop].btnJogPositive THEN
						arrAxisState[iSelectedAxisPageIndex][iLoop] := VISU_CTRL_AXIS_JOG_POSITIVE;
						
					ELSIF arrAxisFrame[iSelectedAxisPageIndex][iLoop].btnJogNegative THEN
						arrAxisState[iSelectedAxisPageIndex][iLoop] := VISU_CTRL_AXIS_JOG_NEGATIVE;
						
					ELSIF arrAxisFrame[iSelectedAxisPageIndex][iLoop].btnAbort THEN
						arrAxisFrame[iSelectedAxisPageIndex][iLoop].btnAbort := FALSE;
						arrAxisState[iSelectedAxisPageIndex][iLoop] := VISU_CTRL_AXIS_ABORT;
						
					END_IF
					
				VISU_CTRL_AXIS_INIT:
					arrAxisLink[iSelectedAxisPageIndex][iLoop].MR_Init();
					
					IF arrAxisLink[iSelectedAxisPageIndex][iLoop].Active THEN
						arrAxisState[iSelectedAxisPageIndex][iLoop] := VISU_CTRL_AXIS_WAIT_FOR_CMD;
					END_IF
				
				VISU_CTRL_AXIS_HOME:
					arrAxisLink[iSelectedAxisPageIndex][iLoop].MR_Home(0.0);
					
					IF arrAxisLink[iSelectedAxisPageIndex][iLoop].IsHomed THEN
						arrAxisState[iSelectedAxisPageIndex][iLoop] := VISU_CTRL_AXIS_WAIT_FOR_CMD;
					END_IF
				
				VISU_CTRL_AXIS_RESET:
					arrAxisLink[iSelectedAxisPageIndex][iLoop].MR_Reset();
					
					IF NOT arrAxisLink[iSelectedAxisPageIndex][iLoop].Error AND NOT arrAxisLink[iSelectedAxisPageIndex][iLoop].Busy THEN
						arrAxisState[iSelectedAxisPageIndex][iLoop] := VISU_CTRL_AXIS_WAIT_FOR_CMD;
					END_IF
				
				VISU_CTRL_AXIS_JOG_POSITIVE:
					arrAxisLink[iSelectedAxisPageIndex][iLoop].JogDirection := E_AxisJogDirection.AXIS_JOG_DIR_POSITIVE;													
					arrAxisLink[iSelectedAxisPageIndex][iLoop].MR_Jog(bJogActive := arrAxisFrame[iSelectedAxisPageIndex][iLoop].btnJogPositive);
					
					IF arrAxisLink[iSelectedAxisPageIndex][iLoop].JogDone THEN
						arrAxisState[iSelectedAxisPageIndex][iLoop] := VISU_CTRL_AXIS_WAIT_FOR_CMD;
					END_IF
				
				VISU_CTRL_AXIS_JOG_NEGATIVE:
					arrAxisLink[iSelectedAxisPageIndex][iLoop].JogDirection := E_AxisJogDirection.AXIS_JOG_DIR_NEGATIVE;														
					arrAxisLink[iSelectedAxisPageIndex][iLoop].MR_Jog(bJogActive := arrAxisFrame[iSelectedAxisPageIndex][iLoop].btnJogNegative);
										
					IF arrAxisLink[iSelectedAxisPageIndex][iLoop].JogDone THEN
						arrAxisState[iSelectedAxisPageIndex][iLoop] := VISU_CTRL_AXIS_WAIT_FOR_CMD;
					END_IF
				
				VISU_CTRL_AXIS_HALT:
					arrAxisLink[iSelectedAxisPageIndex][iLoop].MR_Halt();
					
					IF arrAxisLink[iSelectedAxisPageIndex][iLoop].Halted THEN
						arrAxisState[iSelectedAxisPageIndex][iLoop] := VISU_CTRL_AXIS_WAIT_FOR_CMD;
					END_IF	
				
				VISU_CTRL_AXIS_ABORT:
					arrAxisLink[iSelectedAxisPageIndex][iLoop].MR_Abort();
					
					IF NOT arrAxisLink[iSelectedAxisPageIndex][iLoop].Active THEN
						arrAxisState[iSelectedAxisPageIndex][iLoop] := VISU_CTRL_AXIS_WAIT_FOR_CMD;
					END_IF
				
			END_CASE
			
			(* Check if next frame is empty and exit loop *)
			IF arrAxisFrameEmpty[iSelectedAxisPageIndex][iLoop + 1] = TRUE THEN
				EXIT;
			END_IF
		END_IF
	END_FOR
END_IF
END_METHOD

METHOD PROTECTED MS_ManualCylinders
VAR_INPUT
END_VAR
eCurrentScreen := SCREEN_MANUAL_CYLINDERS;

MS_Manual();

IF arrCylinderFrameEmpty[iCylinderPageIndex][0] THEN
	iCylinderPageIndex := iCylinderPageIndex - 1;
END_IF

bNextInvisible := iSelectedCylinderPageIndex = iCylinderPageIndex;
bPreviousInvisible := iSelectedCylinderPageIndex = 0;

(* Frames control *)
IF btnPrevious THEN
	btnPrevious := FALSE;
	iSelectedCylinderPageIndex := iSelectedCylinderPageIndex - 1;
ELSIF btnNext THEN
	btnNext := FALSE;
	iSelectedCylinderPageIndex := iSelectedCylinderPageIndex + 1;
END_IF

IF iCylinderIndex > 0 THEN
	FOR iLoop := 0 TO iCYLINDERS_PER_PAGE-1 DO
		IF arrCylinderFrameEmpty[iSelectedCylinderPageIndex][iLoop] = FALSE THEN
			arrCylinderFrame[iSelectedCylinderPageIndex][iLoop].bSensorActive := arrCylinderLink[iSelectedCylinderPageIndex][iLoop].PositionActive;
			arrCylinderFrame[iSelectedCylinderPageIndex][iLoop].bSensorHome := arrCylinderLink[iSelectedCylinderPageIndex][iLoop].PositionHome;
			arrCylinderFrame[iSelectedCylinderPageIndex][iLoop].bPositionHold := arrCylinderLink[iSelectedCylinderPageIndex][iLoop].PositionHold;
			arrCylinderFrame[iSelectedCylinderPageIndex][iLoop].bError := arrCylinderLink[iSelectedCylinderPageIndex][iLoop].Error;
			arrCylinderFrame[iSelectedCylinderPageIndex][iLoop].iErrorID := arrCylinderLink[iSelectedCylinderPageIndex][iLoop].ErrorID;
			arrCylinderFrame[iSelectedCylinderPageIndex][iLoop].eCylinderState := arrCylinderLink[iSelectedCylinderPageIndex][iLoop].State;
			arrCylinderFrame[iSelectedCylinderPageIndex][iLoop].sName := arrCylinderLink[iSelectedCylinderPageIndex][iLoop].Name;
			arrCylinderFrame[iSelectedCylinderPageIndex][iLoop].tActiveMovement := arrCylinderLink[iSelectedCylinderPageIndex][iLoop].MoveActiveTime;
			arrCylinderFrame[iSelectedCylinderPageIndex][iLoop].tHomeMovement := arrCylinderLink[iSelectedCylinderPageIndex][iLoop].MoveHomeTime;
			
			(* Requests handling *)
			IF arrCylinderFrame[iSelectedCylinderPageIndex][iLoop].btnReset THEN
				arrCylinderState[iSelectedCylinderPageIndex][iLoop] := VISU_CTRL_CYLINDER_RESET;
			END_IF
			
			CASE arrCylinderState[iSelectedCylinderPageIndex][iLoop] OF
				VISU_CTRL_CYLINDER_WAIT_FOR_CMD:
					IF arrCylinderFrame[iSelectedCylinderPageIndex][iLoop].btnInit THEN
						arrCylinderState[iSelectedCylinderPageIndex][iLoop] := VISU_CTRL_CYLINDER_INIT;
						
					ELSIF arrCylinderFrame[iSelectedCylinderPageIndex][iLoop].btnGoHome THEN
						arrCylinderState[iSelectedCylinderPageIndex][iLoop] := VISU_CTRL_CYLINDER_GO_HOME;
						
					ELSIF arrCylinderFrame[iSelectedCylinderPageIndex][iLoop].btnGoActive THEN
						arrCylinderState[iSelectedCylinderPageIndex][iLoop] := VISU_CTRL_CYLINDER_GO_ACTIVE;
						
					ELSIF arrCylinderFrame[iSelectedCylinderPageIndex][iLoop].btnRealase THEN
						arrCylinderState[iSelectedCylinderPageIndex][iLoop] := VISU_CTRL_CYLINDER_GO_RELEASE;
						
					ELSIF arrCylinderFrame[iSelectedCylinderPageIndex][iLoop].btnAbort THEN
						arrCylinderState[iSelectedCylinderPageIndex][iLoop] := VISU_CTRL_CYLINDER_ABORT;
						
					END_IF
					
				VISU_CTRL_CYLINDER_INIT:
					arrCylinderLink[iSelectedCylinderPageIndex][iLoop].MR_Init();
					
					IF arrCylinderLink[iSelectedCylinderPageIndex][iLoop].Active THEN
						arrCylinderState[iSelectedCylinderPageIndex][iLoop] := VISU_CTRL_CYLINDER_WAIT_FOR_CMD;
					END_IF
					
				VISU_CTRL_CYLINDER_RESET:
					arrCylinderLink[iSelectedCylinderPageIndex][iLoop].MR_Reset();
					
					IF NOT arrCylinderLink[iSelectedCylinderPageIndex][iLoop].Error THEN
						arrCylinderState[iSelectedCylinderPageIndex][iLoop] := VISU_CTRL_CYLINDER_WAIT_FOR_CMD;
					END_IF
				
				VISU_CTRL_CYLINDER_GO_HOME:
					arrCylinderLink[iSelectedCylinderPageIndex][iLoop].MR_GoHome();
					arrCylinderFrame[iSelectedCylinderPageIndex][iLoop].sHomeDescription := arrCylinderFrame[iSelectedCylinderPageIndex][iLoop].sHomeDescription;
					
					IF arrCylinderLink[iSelectedCylinderPageIndex][iLoop].PositionHome AND NOT arrCylinderLink[iSelectedCylinderPageIndex][iLoop].Busy THEN
						arrCylinderState[iSelectedCylinderPageIndex][iLoop] := VISU_CTRL_CYLINDER_WAIT_FOR_CMD;
					END_IF
				
				VISU_CTRL_CYLINDER_GO_ACTIVE:
					arrCylinderLink[iSelectedCylinderPageIndex][iLoop].MR_GoActive();
					arrCylinderFrame[iSelectedCylinderPageIndex][iLoop].sActiveDescription := arrCylinderFrame[iSelectedCylinderPageIndex][iLoop].sActiveDescription;
					
					IF arrCylinderLink[iSelectedCylinderPageIndex][iLoop].PositionActive AND NOT arrCylinderLink[iSelectedCylinderPageIndex][iLoop].Busy THEN
						arrCylinderState[iSelectedCylinderPageIndex][iLoop] := VISU_CTRL_CYLINDER_WAIT_FOR_CMD;
					END_IF
				
				VISU_CTRL_CYLINDER_GO_RELEASE:
					arrCylinderLink[iSelectedCylinderPageIndex][iLoop].MR_Release();
					
					IF NOT arrCylinderLink[iSelectedCylinderPageIndex][iLoop].PositionHold THEN
						arrCylinderState[iSelectedCylinderPageIndex][iLoop] := VISU_CTRL_CYLINDER_WAIT_FOR_CMD;
					END_IF
					
				VISU_CTRL_CYLINDER_ABORT:
					arrCylinderLink[iSelectedCylinderPageIndex][iLoop].MR_Abort();
					
					IF NOT arrCylinderLink[iSelectedCylinderPageIndex][iLoop].Active THEN
						arrCylinderState[iSelectedCylinderPageIndex][iLoop] := VISU_CTRL_CYLINDER_WAIT_FOR_CMD;
					END_IF
				
			END_CASE
			(* Check if next frame is empty and exit loop *)
			IF arrCylinderFrameEmpty[iSelectedCylinderPageIndex][iLoop + 1] = TRUE THEN
				EXIT;
			END_IF
		END_IF
	END_FOR
END_IF
END_METHOD

METHOD PROTECTED MS_ManualInputs
VAR_INPUT
END_VAR
eCurrentScreen := SCREEN_MANUAL_INPUTS;

MS_Manual();

IF arrInputFrameEmpty[iInputPageIndex][0] THEN
	iInputPageIndex := iInputPageIndex - 1;
END_IF

bNextInvisible := iSelectedInputPageIndex = iInputPageIndex;
bPreviousInvisible := iSelectedInputPageIndex = 0;

(* Frames control *)
IF btnPrevious THEN
	btnPrevious := FALSE;
	iSelectedInputPageIndex := iSelectedInputPageIndex - 1;
ELSIF btnNext THEN
	btnNext := FALSE;
	iSelectedInputPageIndex := iSelectedInputPageIndex + 1;
END_IF

IF iInputIndex > 0 THEN
	FOR iLoop := 0 TO iINPUTS_PER_PAGE-1 DO
		IF arrInputFrameEmpty[iSelectedInputPageIndex][iLoop] = FALSE THEN
			arrInputFrame[iSelectedInputPageIndex][iLoop].sName := arrInputLink[iSelectedInputPageIndex][iLoop].Name;
			arrInputFrame[iSelectedInputPageIndex][iLoop].sModuleType := arrInputLink[iSelectedInputPageIndex][iLoop].ModuleType;
			arrInputFrame[iSelectedInputPageIndex][iLoop].sPortID := arrInputLink[iSelectedInputPageIndex][iLoop].PortID;
			arrInputFrame[iSelectedInputPageIndex][iLoop].bIn := arrInputLink[iSelectedInputPageIndex][iLoop].In;
			
			arrInputLink[iSelectedInputPageIndex][iLoop].EnableForce := NOT(arrInputFrame[iSelectedInputPageIndex][iLoop].bForceDisabled);
			
			IF arrInputFrame[iSelectedInputPageIndex][iLoop].bForceIn THEN
				arrInputLink[iSelectedInputPageIndex][iLoop].MR_SetForceValue();
			ELSE 
				arrInputLink[iSelectedInputPageIndex][iLoop].MR_ResetForceValue();
			END_IF
			
			IF arrInputFrameEmpty[iSelectedInputPageIndex][iLoop + 1] = TRUE THEN
				EXIT;
			END_IF
		END_IF
	END_FOR
END_IF
END_METHOD

METHOD PROTECTED MS_ManualOthers
VAR_INPUT
END_VAR
eCurrentScreen := SCREEN_MANUAL_OTHERS;

MS_Manual();
END_METHOD

METHOD PROTECTED MS_ManualOutputs
VAR_INPUT
END_VAR
eCurrentScreen := SCREEN_MANUAL_OUTPUTS;

MS_Manual();

IF arrOutputFrameEmpty[iOutputPageIndex][0] THEN
	iOutputPageIndex := iOutputPageIndex - 1;
END_IF

bNextInvisible := iSelectedOutputPageIndex = iOutputPageIndex;
bPreviousInvisible := iSelectedOutputPageIndex = 0;

(* Frames control *)
IF btnPrevious THEN
	btnPrevious := FALSE;
	iSelectedOutputPageIndex := iSelectedOutputPageIndex - 1;
ELSIF btnNext THEN
	btnNext := FALSE;
	iSelectedOutputPageIndex := iSelectedOutputPageIndex + 1;
END_IF

IF iOutputIndex > 0 THEN
	FOR iLoop := 0 TO iOUTPUTS_PER_PAGE-1 DO
		IF arrOutputFrameEmpty[iSelectedOutputPageIndex][iLoop] = FALSE THEN
			//arrOutputFrame[iSelectedOutputPageIndex][iLoop].bControlable := arrOutputLink[iSelectedOutputPageIndex][iLoop].;
			arrOutputFrame[iSelectedOutputPageIndex][iLoop].sName := arrOutputLink[iSelectedOutputPageIndex][iLoop].Name;
			arrOutputFrame[iSelectedOutputPageIndex][iLoop].sModuleType := arrOutputLink[iSelectedOutputPageIndex][iLoop].ModuleType;
			arrOutputFrame[iSelectedOutputPageIndex][iLoop].sPortID := arrOutputLink[iSelectedOutputPageIndex][iLoop].PortID;
			arrOutputFrame[iSelectedOutputPageIndex][iLoop].bOut := arrOutputLink[iSelectedOutputPageIndex][iLoop].Out;
			
			(* Controll output *)
			arrOutputLink[iSelectedOutputPageIndex][iLoop].Out := arrOutputFrame[iSelectedOutputPageIndex][iLoop].btnOut;
			IF arrOutputFrameEmpty[iSelectedOutputPageIndex][iLoop +1 ] = TRUE THEN
				EXIT;
			END_IF
		END_IF
	END_FOR
END_IF
END_METHOD

METHOD PROTECTED MS_ManualRobots
VAR_INPUT
END_VAR
eCurrentScreen := SCREEN_MANUAL_ROBOTS;

MS_Manual();

IF arrRobotFrameEmpty[iRobotPageIndex][0] THEN
	iRobotPageIndex := iRobotPageIndex - 1;
END_IF

bNextInvisible := iSelectedRobotPageIndex = iRobotPageIndex;
bPreviousInvisible := iSelectedRobotPageIndex = 0;



(* Frames control *)
IF btnPrevious THEN
	btnPrevious := FALSE;
	iSelectedRobotPageIndex := iSelectedRobotPageIndex - 1;
ELSIF btnNext THEN
	btnNext := FALSE;
	iSelectedRobotPageIndex := iSelectedRobotPageIndex + 1;
END_IF

IF iRobotIndex > 0 THEN
	FOR iLoop := 0 TO iROBOTS_PER_PAGE-1 DO
		IF arrRobotFrameEmpty[iSelectedRobotPageIndex][iLoop] = FALSE THEN
			arrRobotFrame[iSelectedRobotPageIndex][iLoop].bIsHomed := arrRobotLink[iSelectedRobotPageIndex][iLoop].IsHomed;
			arrRobotFrame[iSelectedRobotPageIndex][iLoop].bInit := arrRobotLink[iSelectedRobotPageIndex][iLoop].Active;			
			arrRobotFrame[iSelectedRobotPageIndex][iLoop].bError := arrRobotLink[iSelectedRobotPageIndex][iLoop].Error;
			arrRobotFrame[iSelectedRobotPageIndex][iLoop].sErrorDescription := arrRobotLink[iSelectedRobotPageIndex][iLoop].ErrorName;
			arrRobotFrame[iSelectedRobotPageIndex][iLoop].eRobotState := arrRobotLink[iSelectedRobotPageIndex][iLoop].State;
			arrRobotFrame[iSelectedRobotPageIndex][iLoop].sName := arrRobotLink[iSelectedRobotPageIndex][iLoop].Name;
			arrRobotFrame[iSelectedRobotPageIndex][iLoop].bServoOff := arrRobotLink[iSelectedRobotPageIndex][iLoop].ServoIsOff;
			arrRobotFrame[iSelectedRobotPageIndex][iLoop].bServoOn := arrRobotLink[iSelectedRobotPageIndex][iLoop].ServoIsOn;
			arrRobotFrame[iSelectedRobotPageIndex][iLoop].bPaused := arrRobotLink[iSelectedRobotPageIndex][iLoop].Pausing;
			arrRobotFrame[iSelectedRobotPageIndex][iLoop].bStopped := arrRobotLink[iSelectedRobotPageIndex][iLoop].ProgramStopped;
			arrRobotFrame[iSelectedRobotPageIndex][iLoop].bStarted := arrRobotLink[iSelectedRobotPageIndex][iLoop].DoingAction;
			arrRobotFrame[iSelectedRobotPageIndex][iLoop].bPowerOn := arrRobotLink[iSelectedRobotPageIndex][iLoop].CR800PoweredOn;			
			arrRobotFrame[iSelectedRobotPageIndex][iLoop].bBatteryLow := arrRobotLink[iSelectedRobotPageIndex][iLoop].BatteryLow;	
			arrRobotFrame[iSelectedRobotPageIndex][iLoop].bUninitialized := arrRobotLink[iSelectedRobotPageIndex][iLoop].Uninitialized;			
			
			(* Assign parameters from frame to object *)
			arrRobotLink[iSelectedRobotPageIndex][iLoop].ActionNumber := arrRobotFrame[iSelectedRobotPageIndex][iLoop].iActionNumber;
			arrRobotLink[iSelectedRobotPageIndex][iLoop].Override := arrRobotFrame[iSelectedRobotPageIndex][iLoop].iOverride;
			
			(* Assigning state of button disable *)
			arrRobotFrame[iSelectedRobotPageIndex][iLoop].bModeSwitchButtonDisabled := bModeSwitchButtonDisabled;
						
			IF arrRobotLink[iSelectedRobotPageIndex][iLoop].Uninitialized OR arrRobotLink[iSelectedRobotPageIndex][iLoop].AutoModeStarted OR NOT arrRobotLink[iSelectedRobotPageIndex][iLoop].IsHomed THEN
				arrRobotFrame[iSelectedRobotPageIndex][iLoop].bAutoButtonDisable := TRUE;
			ELSE
				arrRobotFrame[iSelectedRobotPageIndex][iLoop].bAutoButtonDisable := FALSE;
			END_IF

			IF arrRobotLink[iSelectedRobotPageIndex][iLoop].Uninitialized OR arrRobotLink[iSelectedRobotPageIndex][iLoop].IsHomed THEN
				arrRobotFrame[iSelectedRobotPageIndex][iLoop].bHomeButtonDisable := TRUE;
			ELSE
				arrRobotFrame[iSelectedRobotPageIndex][iLoop].bHomeButtonDisable := FALSE;
			END_IF
			
			IF arrRobotLink[iSelectedRobotPageIndex][iLoop].Uninitialized OR NOT arrRobotLink[iSelectedRobotPageIndex][iLoop].AutoModeStarted OR arrRobotLink[iSelectedRobotPageIndex][iLoop].DoingAction OR arrRobotLink[iSelectedRobotPageIndex][iLoop].Pausing OR arrRobotLink[iSelectedRobotPageIndex][iLoop].ProgramStopped THEN
				arrRobotFrame[iSelectedRobotPageIndex][iLoop].bActionButtonDisable := TRUE;
			ELSE
				arrRobotFrame[iSelectedRobotPageIndex][iLoop].bActionButtonDisable := FALSE;
			END_IF

			IF arrRobotLink[iSelectedRobotPageIndex][iLoop].Uninitialized OR NOT arrRobotLink[iSelectedRobotPageIndex][iLoop].DoingAction OR arrRobotLink[iSelectedRobotPageIndex][iLoop].Pausing OR arrRobotLink[iSelectedRobotPageIndex][iLoop].ProgramStopped THEN
				arrRobotFrame[iSelectedRobotPageIndex][iLoop].bPausingButtonDisable := TRUE;
			ELSE
				arrRobotFrame[iSelectedRobotPageIndex][iLoop].bPausingButtonDisable := FALSE;
			END_IF
			
			IF arrRobotLink[iSelectedRobotPageIndex][iLoop].Uninitialized OR NOT arrRobotLink[iSelectedRobotPageIndex][iLoop].Pausing OR arrRobotLink[iSelectedRobotPageIndex][iLoop].ProgramStopped THEN
				arrRobotFrame[iSelectedRobotPageIndex][iLoop].bRestoreCycleButtonDisable := TRUE;
			ELSE
				arrRobotFrame[iSelectedRobotPageIndex][iLoop].bRestoreCycleButtonDisable := FALSE;
			END_IF	

			IF arrRobotLink[iSelectedRobotPageIndex][iLoop].Uninitialized OR NOT arrRobotLink[iSelectedRobotPageIndex][iLoop].DoingAction OR arrRobotLink[iSelectedRobotPageIndex][iLoop].ProgramStopped OR arrRobotLink[iSelectedRobotPageIndex][iLoop].Pausing THEN
				arrRobotFrame[iSelectedRobotPageIndex][iLoop].bStoppingButtonDisable := TRUE;
			ELSE
				arrRobotFrame[iSelectedRobotPageIndex][iLoop].bStoppingButtonDisable := FALSE;
			END_IF	
			
			IF arrRobotLink[iSelectedRobotPageIndex][iLoop].Uninitialized OR NOT arrRobotLink[iSelectedRobotPageIndex][iLoop].ProgramStopped OR arrRobotLink[iSelectedRobotPageIndex][iLoop].Pausing THEN
				arrRobotFrame[iSelectedRobotPageIndex][iLoop].bRestoreAutoButtonDisable := TRUE;
			ELSE
				arrRobotFrame[iSelectedRobotPageIndex][iLoop].bRestoreAutoButtonDisable := FALSE;
			END_IF	
		
			(* Requests handling *)
			IF arrRobotFrame[iSelectedRobotPageIndex][iLoop].btnErrorReset THEN
				arrRobotState[iSelectedRobotPageIndex][iLoop] := VISU_CTRL_ROBOT_ERR_RESET;
			END_IF
			
			(* Requests handling *)
			IF arrRobotFrame[iSelectedRobotPageIndex][iLoop].btnControllerReset THEN
				arrRobotState[iSelectedRobotPageIndex][iLoop] := VISU_CTRL_ROBOT_CONTROLLER_RESET;
			END_IF
			
			(* Requests handling *)
			IF arrRobotFrame[iSelectedRobotPageIndex][iLoop].btnAbort THEN
				arrRobotState[iSelectedRobotPageIndex][iLoop] := VISU_CTRL_ROBOT_ABORT;
			END_IF
			
			IF arrRobotFrame[iSelectedRobotPageIndex][iLoop].btnCyclePause THEN
				arrRobotState[iSelectedRobotPageIndex][iLoop] := VISU_CTRL_ROBOT_CYCLE_PAUSE;
			END_IF			
			
			IF arrRobotFrame[iSelectedRobotPageIndex][iLoop].btnCycleStop THEN
				arrRobotState[iSelectedRobotPageIndex][iLoop] := VISU_CTRL_ROBOT_CYCLE_STOP;
			END_IF	
	
			CASE arrRobotState[iSelectedRobotPageIndex][iLoop] OF
				VISU_CTRL_ROBOT_WAIT_FOR_CMD:
					IF arrRobotFrame[iSelectedRobotPageIndex][iLoop].btnInit THEN
						arrRobotState[iSelectedRobotPageIndex][iLoop] := VISU_CTRL_ROBOT_INIT;
						
					ELSIF arrRobotFrame[iSelectedRobotPageIndex][iLoop].btnGoHome THEN
						arrRobotState[iSelectedRobotPageIndex][iLoop] := VISU_CTRL_ROBOT_GO_HOME;
						
					ELSIF arrRobotFrame[iSelectedRobotPageIndex][iLoop].btnDoAction THEN
						arrRobotState[iSelectedRobotPageIndex][iLoop] := VISU_CTRL_ROBOT_DO_ACTION;
						
					ELSIF arrRobotFrame[iSelectedRobotPageIndex][iLoop].btnUpdateRecipes THEN
						arrRobotState[iSelectedRobotPageIndex][iLoop] := VISU_CTRL_ROBOT_UPDATE_RECIPES;
						
					ELSIF arrRobotFrame[iSelectedRobotPageIndex][iLoop].btnGoAuto THEN
						arrRobotState[iSelectedRobotPageIndex][iLoop] := VISU_CTRL_ROBOT_GO_AUTO;
						
					ELSIF arrRobotFrame[iSelectedRobotPageIndex][iLoop].btnRestoreCycle THEN
						arrRobotState[iSelectedRobotPageIndex][iLoop] := VISU_CTRL_ROBOT_RESTORE_CYCLE;
						
					ELSIF arrRobotFrame[iSelectedRobotPageIndex][iLoop].btnRestoreAuto THEN
						arrRobotState[iSelectedRobotPageIndex][iLoop] := VISU_CTRL_ROBOT_RESTORE_AUTO;

					ELSIF arrRobotFrame[iSelectedRobotPageIndex][iLoop].btnBatteryReset THEN
						arrRobotState[iSelectedRobotPageIndex][iLoop] := VISU_CTRL_ROBOT_BATTERY_RESET;
						
					END_IF

					
				VISU_CTRL_ROBOT_INIT:
					arrRobotLink[iSelectedRobotPageIndex][iLoop].MR_Init();
					
					IF arrRobotLink[iSelectedRobotPageIndex][iLoop].Active THEN
						arrRobotState[iSelectedRobotPageIndex][iLoop] := VISU_CTRL_ROBOT_WAIT_FOR_CMD;
					END_IF
					
				VISU_CTRL_ROBOT_ERR_RESET:
					arrRobotLink[iSelectedRobotPageIndex][iLoop].MR_Reset();
					
					IF NOT arrRobotLink[iSelectedRobotPageIndex][iLoop].Busy THEN
						arrRobotState[iSelectedRobotPageIndex][iLoop] := VISU_CTRL_ROBOT_WAIT_FOR_CMD;
					END_IF
				
				VISU_CTRL_ROBOT_CONTROLLER_RESET:
					arrRobotLink[iSelectedRobotPageIndex][iLoop].MR_ResetCR800Err();
					
					IF NOT arrRobotLink[iSelectedRobotPageIndex][iLoop].Busy THEN
						arrRobotState[iSelectedRobotPageIndex][iLoop] := VISU_CTRL_ROBOT_WAIT_FOR_CMD;
					END_IF
				
				VISU_CTRL_ROBOT_ABORT:
					arrRobotLink[iSelectedRobotPageIndex][iLoop].MR_Abort();
					
					IF NOT arrRobotLink[iSelectedRobotPageIndex][iLoop].Active THEN
						arrRobotState[iSelectedRobotPageIndex][iLoop] := VISU_CTRL_ROBOT_WAIT_FOR_CMD;
					END_IF
				
				VISU_CTRL_ROBOT_GO_HOME:
					arrRobotLink[iSelectedRobotPageIndex][iLoop].MR_GoHome();
					
					IF NOT arrRobotLink[iSelectedRobotPageIndex][iLoop].Busy THEN
						arrRobotState[iSelectedRobotPageIndex][iLoop] := VISU_CTRL_ROBOT_WAIT_FOR_CMD;
					END_IF
					
				VISU_CTRL_ROBOT_DO_ACTION:
					arrRobotLink[iSelectedRobotPageIndex][iLoop].MR_DoAction(arrRobotFrame[iSelectedRobotPageIndex][iLoop].iActionNumber);
					
					IF NOT arrRobotLink[iSelectedRobotPageIndex][iLoop].Busy THEN
						arrRobotState[iSelectedRobotPageIndex][iLoop] := VISU_CTRL_ROBOT_WAIT_FOR_CMD;
					END_IF

				VISU_CTRL_ROBOT_UPDATE_RECIPES:
					arrRobotLink[iSelectedRobotPageIndex][iLoop].MR_UpdateRecipies();
					
					IF NOT arrRobotLink[iSelectedRobotPageIndex][iLoop].Busy THEN
						arrRobotState[iSelectedRobotPageIndex][iLoop] := VISU_CTRL_ROBOT_WAIT_FOR_CMD;
					END_IF
			
				VISU_CTRL_ROBOT_GO_AUTO:
					arrRobotLink[iSelectedRobotPageIndex][iLoop].MR_GoAuto();
					
					IF NOT arrRobotLink[iSelectedRobotPageIndex][iLoop].Busy THEN
						arrRobotState[iSelectedRobotPageIndex][iLoop] := VISU_CTRL_ROBOT_WAIT_FOR_CMD;
					END_IF

				VISU_CTRL_ROBOT_CYCLE_PAUSE:
					arrRobotLink[iSelectedRobotPageIndex][iLoop].MR_CyclePause();
					
					IF NOT arrRobotLink[iSelectedRobotPageIndex][iLoop].Busy THEN
						arrRobotState[iSelectedRobotPageIndex][iLoop] := VISU_CTRL_ROBOT_WAIT_FOR_CMD;
					END_IF

				VISU_CTRL_ROBOT_CYCLE_STOP:
					arrRobotLink[iSelectedRobotPageIndex][iLoop].MR_CycleStop();
					
					IF NOT arrRobotLink[iSelectedRobotPageIndex][iLoop].Busy THEN
						arrRobotState[iSelectedRobotPageIndex][iLoop] := VISU_CTRL_ROBOT_WAIT_FOR_CMD;
					END_IF

				VISU_CTRL_ROBOT_RESTORE_CYCLE:
					arrRobotLink[iSelectedRobotPageIndex][iLoop].MR_RestoreCycle();
					
					IF NOT arrRobotLink[iSelectedRobotPageIndex][iLoop].Busy THEN
						arrRobotState[iSelectedRobotPageIndex][iLoop] := VISU_CTRL_ROBOT_WAIT_FOR_CMD;
					END_IF

				VISU_CTRL_ROBOT_RESTORE_AUTO:
					arrRobotLink[iSelectedRobotPageIndex][iLoop].MR_RestoreAuto();
					
					IF NOT arrRobotLink[iSelectedRobotPageIndex][iLoop].Busy THEN
						arrRobotState[iSelectedRobotPageIndex][iLoop] := VISU_CTRL_ROBOT_WAIT_FOR_CMD;
					END_IF
					
				VISU_CTRL_ROBOT_BATTERY_RESET:
					arrRobotLink[iSelectedRobotPageIndex][iLoop].MR_BatteryReset();
					
					IF NOT arrRobotLink[iSelectedRobotPageIndex][iLoop].Busy THEN
						arrRobotState[iSelectedRobotPageIndex][iLoop] := VISU_CTRL_ROBOT_WAIT_FOR_CMD;
					END_IF		
					
			END_CASE
			(* Check if next frame is empty and exit loop *)
			IF arrRobotFrameEmpty[iSelectedRobotPageIndex][iLoop + 1] = TRUE THEN
				EXIT;
			END_IF
		END_IF
	END_FOR
END_IF
END_METHOD

METHOD PROTECTED MS_ManualSafety
VAR_INPUT
END_VAR
eCurrentScreen := SCREEN_MANUAL_SAFETY;

MS_Manual();

IF arrSafeInputFrameEmpty[iSafeInputPageIndex][0] THEN
	iSafeInputPageIndex := iSafeInputPageIndex - 1;
END_IF

bNextInvisibleInput := iSelectedSafeInputPageIndex = iSafeInputPageIndex;
bPreviousInvisibleInput := iSelectedSafeInputPageIndex = 0;

(* Frames control *)
IF btnPreviousInput THEN
	btnPreviousInput := FALSE;
	iSelectedSafeInputPageIndex := iSelectedSafeInputPageIndex - 1;
ELSIF btnNextInput THEN
	btnNextInput := FALSE;
	iSelectedSafeInputPageIndex := iSelectedSafeInputPageIndex + 1;
END_IF

IF iSafeInputIndex > 0 THEN
	FOR iLoop := 0 TO iSAFE_INPUTS_PER_PAGE-1 DO
		IF arrSafeInputFrameEmpty[iSelectedSafeInputPageIndex][iLoop] = FALSE THEN
			arrSafeInputFrame[iSelectedSafeInputPageIndex][iLoop].sName := arrSafeInputLink[iSelectedSafeInputPageIndex][iLoop].Name;
			arrSafeInputFrame[iSelectedSafeInputPageIndex][iLoop].sModuleType := arrSafeInputLink[iSelectedSafeInputPageIndex][iLoop].ModuleType;
			arrSafeInputFrame[iSelectedSafeInputPageIndex][iLoop].sPortID := arrSafeInputLink[iSelectedSafeInputPageIndex][iLoop].PortID;
			arrSafeInputFrame[iSelectedSafeInputPageIndex][iLoop].bIn := arrSafeInputLink[iSelectedSafeInputPageIndex][iLoop].In;
			
			arrSafeInputLink[iSelectedSafeInputPageIndex][iLoop].EnableForce := NOT(arrSafeInputFrame[iSelectedSafeInputPageIndex][iLoop].bForceDisabled);
			
			IF arrSafeInputFrame[iSelectedSafeInputPageIndex][iLoop].bForceIn THEN
				arrSafeInputLink[iSelectedSafeInputPageIndex][iLoop].MR_SetForceValue();
			ELSE 
				arrSafeInputLink[iSelectedSafeInputPageIndex][iLoop].MR_ResetForceValue();
			END_IF
			
			IF arrSafeInputFrameEmpty[iSelectedSafeInputPageIndex][iLoop + 1] = TRUE THEN
				EXIT;
			END_IF
		END_IF
	END_FOR
END_IF

IF arrSafeOutputFrameEmpty[iSafeOutputPageIndex][0] THEN
	iSafeOutputPageIndex := iSafeOutputPageIndex - 1;
END_IF

bNextInvisibleOutput := iSelectedSafeOutputPageIndex = iSafeOutputPageIndex;
bPreviousInvisibleOutput := iSelectedSafeOutputPageIndex = 0;

(* Frames control *)
IF btnPreviousOutput THEN
	btnPreviousOutput := FALSE;
	iSelectedSafeOutputPageIndex := iSelectedSafeOutputPageIndex - 1;
ELSIF btnNextOutput THEN
	btnNextOutput := FALSE;
	iSelectedSafeOutputPageIndex := iSelectedSafeOutputPageIndex + 1;
END_IF


IF iSafeOutputIndex > 0 THEN
	FOR iLoop := 0 TO iSAFE_OUTPUTS_PER_PAGE-1 DO
		IF arrSafeOutputFrameEmpty[iSelectedOutputPageIndex][iLoop] = FALSE THEN
			//arrOutputFrame[iSelectedOutputPageIndex][iLoop].bControlable := arrOutputLink[iSelectedOutputPageIndex][iLoop].;
			arrSafeOutputFrame[iSelectedSafeOutputPageIndex][iLoop].sName := arrSafeOutputLink[iSelectedSafeOutputPageIndex][iLoop].Name;
			arrSafeOutputFrame[iSelectedSafeOutputPageIndex][iLoop].sModuleType := arrSafeOutputLink[iSelectedSafeOutputPageIndex][iLoop].ModuleType;
			arrSafeOutputFrame[iSelectedSafeOutputPageIndex][iLoop].sPortID := arrSafeOutputLink[iSelectedSafeOutputPageIndex][iLoop].PortID;
			arrSafeOutputFrame[iSelectedSafeOutputPageIndex][iLoop].bOut := arrSafeOutputLink[iSelectedSafeOutputPageIndex][iLoop].Out;
			
			(* Controll output *)
			arrSafeOutputLink[iSelectedSafeOutputPageIndex][iLoop].Out := arrSafeOutputFrame[iSelectedSafeOutputPageIndex][iLoop].btnOut;
			IF arrSafeOutputFrameEmpty[iSelectedSafeOutputPageIndex][iLoop +1 ] = TRUE THEN
				EXIT;
			END_IF
		END_IF
	END_FOR
END_IF
END_METHOD

METHOD PROTECTED MS_ModeChange
VAR_INPUT
END_VAR
eCurrentNavigation := NAVIGATION_EMPTY;

IF ifUniversalMachineLink.State = MACHINE_STATE_AUTO THEN
	eCurrentScreen := SCREEN_AUTO;	
	
ELSIF ifUniversalMachineLink.State = MACHINE_STATE_MANUAL THEN	
	eCurrentScreen := SCREEN_MANUAL_MOTORS;
	
ELSIF ifUniversalMachineLink.State = MACHINE_STATE_EMERGENCY THEN
	eCurrentScreen := SCREEN_EMERGENCY;
	
END_IF
END_METHOD

METHOD PROTECTED MS_ReadyInitialized
VAR_INPUT
END_VAR
eCurrentNavigation := NAVIGATION_INITIALIZING;

IF ifUniversalMachineLink.State = MACHINE_STATE_ABORTING THEN
	eCurrentScreen := SCREEN_ABORTING;	
			
ELSIF ifUniversalMachineLink.State = MACHINE_STATE_AUTO THEN
	eCurrentScreen := SCREEN_AUTO;
	
ELSIF ifUniversalMachineLink.State = MACHINE_STATE_EMERGENCY THEN
	eCurrentScreen := SCREEN_EMERGENCY;
			
END_IF
END_METHOD

METHOD PROTECTED MS_Recipes
VAR_INPUT
END_VAR
eCurrentNavigation := NAVIGATION_UTILITIES;

IF btnBack THEN
	btnBack := FALSE;
	eCurrentScreen := eLastScreen;
	
END_IF

IF arrRobotFrameEmpty[iRecipeParameterPageIndex][0] THEN
	iRecipeParameterPageIndex := iRecipeParameterPageIndex - 1;
END_IF

bRecipeNextInvisible := iSelectedRecipeParameterPageIndex = iRecipeParameterPageIndex;
bRecipePreviousInvisible := iSelectedRecipeParameterPageIndex = 0;

(* Frames control *)
IF btnPrevious THEN
	btnPrevious := FALSE;
	iSelectedRecipeParameterPageIndex := iSelectedRecipeParameterPageIndex - 1;
	
ELSIF btnNext THEN
	btnNext := FALSE;
	iSelectedRecipeParameterPageIndex := iSelectedRecipeParameterPageIndex + 1;
	
END_IF
END_METHOD

METHOD PROTECTED MS_Reset
VAR_INPUT
END_VAR
eCurrentNavigation := NAVIGATION_INITIALIZING;

IF ifUniversalMachineLink.State = MACHINE_STATE_RESET THEN
	eCurrentScreen := SCREEN_RESET;
	
ELSIF ifUniversalMachineLink.State = MACHINE_STATE_RESET_DONE THEN
	eCurrentScreen := SCREEN_AUTO;
	
ELSIF ifUniversalMachineLink.State = MACHINE_STATE_EMERGENCY THEN
	eCurrentScreen := SCREEN_EMERGENCY;
	
END_IF
END_METHOD

METHOD PROTECTED MS_Uninitialized
VAR_INPUT
END_VAR
eCurrentNavigation := NAVIGATION_UNINITIALIZED;

IF ifUniversalMachineLink.State = MACHINE_STATE_INITIALIZING THEN
	eCurrentScreen := SCREEN_INITIALIZING;	
	
END_IF
END_METHOD

PROPERTY Start : REFERENCE TO BOOL
GET
Start REF= btnStart;
END_GET
END_PROPERTY

METHOD PROTECTED StateMachine
VAR_INPUT
END_VAR
CASE eCurrentScreen OF
	SCREEN_UNINITIALIZED:
		MS_Uninitialized();
	
	SCREEN_INITIALIZING:
		MS_Initializing();
		
	SCREEN_READY_INITIALIZED:
		MS_ReadyInitialized();
		
	SCREEN_AUTO:
		MS_Auto();
		
	SCREEN_MODE_CHANGE:
		MS_ModeChange();
	
	SCREEN_MANUAL_CYLINDERS:
		MS_ManualCylinders();
		
	SCREEN_MANUAL_MOTORS:
		MS_ManualAxis();
	
//	SCREEN_MANUAL_SAFETY:
//		MS_ManualSafety();
	
	SCREEN_MANUAL_INPUTS:
		MS_ManualInputs();
	
	SCREEN_MANUAL_OUTPUTS:
		MS_ManualOutputs();
		
	SCREEN_MANUAL_ROBOTS:
		MS_ManualRobots();		
		
	SCREEN_MANUAL_OTHERS:
		MS_ManualOthers();
	
	SCREEN_ALARMS:
		MS_Alarms();
	
	SCREEN_RECIPES:
		MS_Recipes();
		
	SCREEN_RESET:
		MS_Reset();
		
	SCREEN_ABORTING:
		MS_Aborting();
		
	SCREEN_EMERGENCY:
		MS_Emergency();
	
END_CASE
END_METHOD

PROPERTY Stop : REFERENCE TO BOOL
GET
Stop REF= btnStop;
END_GET
END_PROPERTY

END_FUNCTION_BLOCK

// ---- POUs/PRG/PRG_AlarmControl.TcPOU
PROGRAM PRG_AlarmControl
VAR CONSTANT
	sDEFAULT_NAME		: STRING := 'TwinCAT3 Event Logger';	
	sDEFAULT_FILE_PATH	: STRING := 'C:\TcEvents\';
END_VAR
VAR
	bFirstCycle			: BOOL := TRUE;
	fbAlarmControler 	: FB_AlarmControler;
	
	bInit 				: BOOL;
	bAbort				: BOOL;
END_VAR

IF bFirstCycle THEN
	bFirstCycle := FALSE;
	
	fbAlarmControler.MR_FirstCycle( sName		:= sDEFAULT_NAME,
									sFileName	:= sDEFAULT_FILE_PATH);
									
	(* Assign machine controler reference to Shell API*)
	stShell.stPlatform.ref_fbAlarmControler REF= fbAlarmControler;
	
	(* Set assignamnet done bit for visu controler *)
	stShell.stFlags.bAlarmCtrlAssignamentsDone := TRUE;
END_IF

fbAlarmControler();

END_PROGRAM

// ---- POUs/PRG/PRG_MachineControl.TcPOU
(* =======================================================================================================================================
   Automatic Optical Inspection Machine Program
   =======================================================================================================================================
   References
   ======================================================================================================================================= *)
PROGRAM PRG_MachineControl
VAR
	bFirstCycle 		: BOOL := TRUE;			(*  *)
	fbMachineControler 	: FB_MachineControl;	(*  *)
	fbFileLogger 		: FB_FileLogger;		(*	*)
END_VAR

IF bFirstCycle THEN
	bFirstCycle := FALSE;
	
	(* Assign machine controler reference to Shell API*)
	stShell.stPlatform.ref_fbMachineControler REF= fbMachineControler;
	
	(* Set assignamnet done bit for visu controler *)
	stShell.stFlags.bMachineCtrlAssignamentsDone := TRUE;
	
	fbMachineLogger.MR_FirstCycle( 	sName		:= 'AOI_Machine_Logger',
									sFileDir 	:= 'C:\TwinCAT\Loggers',
									sFileName 	:= 'AOI_Machine_Logger',
									sAmsNetId 	:= '',
									bAddTimeStamp := FALSE,
									bAddHeader := FALSE);
END_IF

IF NOT fbMachineLogger.Active THEN 
	fbMachineLogger.MR_Init();	
END_IF
// =========================================================
(* Run global machine clock *)
fbMachineTime(bEnable := TRUE);
(* Cyclic run of machine controler *)
fbMachineControler();
(* Machine Logger *)
fbMachineLogger();
// =========================================================

END_PROGRAM

// ---- POUs/Machine/FB_MachineControl.TcPOU
FUNCTION_BLOCK FB_MachineControl EXTENDS FB_UniversalMachine IMPLEMENTS I_MachineControl
VAR PERSISTENT
	sLastLoadedRecipe						: STRING;
	sLastProductOrder						: STRING;
	(* Parameter have to adjust for Sorting Station *)
	lrSortGoodDistance			: LREAL := -24.0;	(* Distance between cam7 to sort station *)
	lrSortDirtDistance			: LREAL := -55.0;	(* Distance between cam7 to sort station *)
	lrSortDentDistance			: LREAL := -55.0;	(* Distance between cam7 to sort station *)
	lrSortRejectDistance		: LREAL := -60.0;	(* Distance between cam7 to sort station *)
	tSortValveGoodTime			: TIME := T#1000MS;		(* During time to shoot sample *)
	tSortValveDirtTime			: TIME := T#2000MS;		(* During time to shoot sample *)
	tSortValveDentTime			: TIME := T#1000MS;		(* During time to shoot sample *)
	tSortValveRejectTime		: TIME := T#1000MS;		(* During time to shoot sample *)
	
	rBowlFeederSetpoint 		: REAL := 60.0;
END_VAR
VAR	
	(* Process data *)
	//{attribute 'OPC.UA.DA' := '1	'}
	stBatchPerformance		: ST_BatchPerformacne; 	(* Data about performance about current proccesed batch *)
	//{attribute 'OPC.UA.DA' := '1	'}                                                          		
	stBatchData				: ST_BatchData;			(* Data about batch that is going to be processed*)

	(*--- Module Interface ---*)
	fbRobot 					: FB_Robot;
	fbRTCVision 				: FB_RTCVision;
	fbBowlFeeder				: FB_BowlFeeder;
	fbRotaryTable				: FB_AxisServo;
	
	(* Utilities *)
	fbPlcUps					: FB_UpsCx51xx;	
	
	(* IO PLC connect *)
	diProductPresenceBowl		: FB_DigitalInput;	(* *)
	diProductPresenceRobot		: FB_DigitalInput;	(* *)	
	
	poDoorLock					: FB_DigitalOutput;			(* Requests all machine lock's to close *)
	poResetButtonLight			: FB_DigitalOutput;			(* Physical reset button attached to door's of electrical cabinet *)
	
	doBlowBowlFeeder			: FB_DigitalOutput;
	doBlowGood					: FB_DigitalOutput;
	doBlowReject				: FB_DigitalOutput;
	doBlowDentContamination		: FB_DigitalOutput;
	doBlowDirtScratch			: FB_DigitalOutput;
	
	doTriggerCam1				: FB_DoubleTrigger;
	doTriggerCam2				: FB_DoubleTrigger;
	doTriggerCam3				: FB_DoubleTrigger;
	doTriggerCam4				: FB_DoubleTrigger;
	doTriggerCam5				: FB_DoubleTrigger;
	doTriggerCam6				: FB_DoubleTrigger;
	doTriggerCam7				: FB_DoubleTrigger;
	
	
	
	(* Auxilary *)
	tonDelay					: TON;				(* Provides any delay into the machine when switching something On/Off *)
	//tonTestDelay	: TON;	(* Delay which allows to see any page changes during tests *)	
	
	(* Parameter *)
	lrHOME_POSTION				: LREAL := 0.0;		(* Homming position *)
	stRotaryTableHomingOptions	: ST_HomingOptions;
	
	(* #ManualToAuto *)             	                                                            		
	//bManualToAutoRotate					: BOOL;																            	
	bStop								: BOOL;	
		
	// =============== State machine ============================================================
	eMachineStateUninitialized						: E_MachineCtrlStateUninitialized;
	eMachineStateInit								: E_MachineCtrlStateInit;
	eMachineStateAuto								: E_MachineCtrlStateAuto;
	eMachineStateAutoAOI							: E_MachineCtrlStateAutoAOI;
	eMachineStateAbort								: E_MachineCtrlStateAbort;
	eMachineStateManualToAuto						: E_MachineCtrlStateManualToAuto;
	
	(* HMI control *)
	btnStartBowl : BOOL;
	btnStopBowl : BOOL;
	
END_VAR

IF bFirstCycle THEN
	(* - bFirstCycle bit reset by parent *)
	(* --- Assign initial parameters for machine objects ---*)
	(* Assign UPS parameters *)
	fbPlcUps.MR_FirstCycle( 	sName 		:= 'PLC UPS',
								sNetID 		:= '',
								iPlcPort 	:= 851,
								tTimeout 	:= DEFAULT_ADS_TIMEOUT);
								
	(* Assign robots *)
	fbRobot.MR_FirstCycle(	sName				:= 'RH-3CRH4018-D-S15',
							iInitialOverride 	:= 3,					//low for testing
							sPLC_NET_ID 		:= '5.127.48.56.2.1',
							iCR800_1_ADDRESS 	:= 1020);
	
	(* Assign rotary table *)
	fbRotaryTable.MR_FirstCycle(	sName				:= sROTARY_TABLE_NAME,
									sMeasurementUnits	:= sROTARY_TABLE_MEASUREMENT_UNIT,
									bModulo				:= FALSE);
									
	fbRotaryTable.Override 			:= 100.0;
	fbRotaryTable.Velocity 			:= 100.0;	//400,325
	fbRotaryTable.Acceleration 		:= 1500.0; //1500,80|600
	fbRotaryTable.Deceleration 		:= 1500.0; //1500,800|600
	fbRotaryTable.Jerk 				:= 6000.0;//6000.0; //15000,8000|

	fbRotaryTable.JogPosition 		:= 0.0;
	fbRotaryTable.JogVelocity 		:= 300.0;
	fbRotaryTable.JogAcceleration 	:= 800.0;
	fbRotaryTable.JogDeceleration 	:= 800.0;
	fbRotaryTable.JogJerk 			:= 800.0;
	fbRotaryTable.StopDeceleration	:= 800.0;
	fbRotaryTable.StopJerk 			:= 8000.0;
	
	stRotaryTableHomingOptions.SearchDirection := Tc2_MC2.MC_Direction.MC_Negative_Direction;
	stRotaryTableHomingOptions.SearchVelocity 	:= 12.0;
	stRotaryTableHomingOptions.SyncDirection 	:= Tc2_MC2.MC_Direction.MC_Positive_Direction;
	stRotaryTableHomingOptions.SyncVelocity	:= 10.0;
	
	fbRotaryTable.HomingMode		:= MC_HomingMode.MC_DefaultHoming;
	fbRotaryTable.HomingOptions 	:= stRotaryTableHomingOptions;

	(* Assign bowl feeder *)
	fbBowlFeeder.MR_FirstCycle(sName := 'Bowl Feeder');
	fbBowlFeeder.Setpoint := 60.0;
	
	(* Assign RTC Vision system *)
	fbRTCVision.MR_FirstCycle(	sCameraName 	:= 'RTC Vision System',
								sClientHost		:= '10.20.254.8',
								sClientAmsNetID := '',
								iClientPort 	:= 23,
								tTimeout 		:= T#15S);
	
	(* Digital I/O *)
	diProductPresenceBowl.MR_FirstCycle(	sName := 'Product presence on bowl at pick point',
											sModuleType := '',
											sPortID := '');
											
	diProductPresenceRobot.MR_FirstCycle(	sName := 'Product presence at robot nozzle',
											sModuleType := '',
											sPortID := '');
									
	poDoorLock.MR_FirstCycle(		sName := 'Door lock station 1',
		                         sModuleType := '',
                                 sPortID := '');
								 
	poResetButtonLight.MR_FirstCycle(	sName := 'Reset Button light station 1',
										sModuleType := '',
										sPortID := '');

END_IF

(* Execute parent implementation *)
SUPER^();

(* --- Cyclic run ---*)
(* Cyclic run robots *)
fbRobot();
(* Cyclic run RTC vision *)
fbRTCVision();
(* Cyclic run bowl feeder *)
fbBowlFeeder();
(* Cyclic run rotary table *)
fbRotaryTable();
(* Utilities *)
fbPlcUps();

PROPERTY BowlFeeder : REFERENCE TO FB_BowlFeeder
GET
BowlFeeder REF= fbBowlFeeder;
END_GET
END_PROPERTY

METHOD PROTECTED GoldenSample : BOOL
VAR_INPUT
END_VAR
;
END_METHOD

METHOD PROTECTED M_AutoProcessing
VAR_INST
	(* Equipment module sequences *)
	BowlFeederProcess : UINT;
	RobotProcess : UINT;
	
	RotaryTableProcess : UINT;
	TableRegister		: UINT;
	
	(* Parameters *)
	bIsRobotAtRotaryTable : BOOL;
	OneStep : LREAL := 10.00;
END_VAR
/// ======================= Bowl feeder process ======================= {{{
CASE BowlFeederProcess OF
	0:
		IF fbBowlFeeder.MR_Start() THEN
			BowlFeederProcess := 10;
		END_IF
		
	10:
		;
		
END_CASE
///}}}
/// ======================= Robot process ======================= {{{
CASE RobotProcess OF
	0://IDLE go bowl
		fbRobot.MR_GoBowl();
		IF NOT fbRobot.Busy THEN
			RobotProcess := 5;
		END_IF
		
	5://Goto input
		IF diProductPresenceBowl.In THEN (* waiting product *)
			fbRobot.MR_GoInputProduct();
			IF NOT fbRobot.Busy THEN
				RobotProcess := 6;
			END_IF
		END_IF
	
	6://robot pick
		fbRobot.MR_Pick();
		IF NOT fbRobot.Busy THEN
			RobotProcess := 10;
		END_IF 
		
	10://go to station 1
		fbRobot.MR_GoStation1();
		IF NOT fbRobot.Busy THEN
			RobotProcess := 20;
		END_IF
	20:
		fbRTCVision.M_CommandStation1(DelayTimeForSecondTrigger := T#1MS);
		IF NOT fbRTCVision.Busy THEN
			RobotProcess := 30;
		END_IF
	30:
		fbRobot.MR_GoStation2();
		IF NOT fbRobot.Busy THEN
			RobotProcess := 40;
		END_IF
	40:
		fbRTCVision.M_CommandStation2(DelayTimeForSecondTrigger := T#34MS);
		IF NOT fbRTCVision.Busy THEN
			RobotProcess := 50;
		END_IF
	50:
		fbrobot.MR_GoRotaryTable();
		IF NOT fbrobot.Busy THEN
			RobotProcess:= 60;//waiting drop product
		END_IF
	
END_CASE

IF RobotProcess = 60 THEN
	bIsRobotAtRotaryTable := TRUE;
ELSE
	bIsRobotAtRotaryTable := FALSE;
END_IF

///}}}
///(*======================= Rotary Table process =======================*){{{
(* Product placed and reset robot sequence *)
CASE TableRegister OF
	0://take product from robot
		IF fbRotaryTable.Halted AND bIsRobotAtRotaryTable THEN
			fbrobot.MR_Place();
			IF NOT fbrobot.Busy THEN
				TableRegister := 10;
			END_IF
		END_IF
	10://buffer calc and add process
		IF Buffer_RotaryTable.Add2Data(in1 := fbRotaryTable.ActualPosition + OneStep, in2 := fbRotaryTable.ActualPosition + 2*OneStep) THEN
			IF Buffer_Station3.Add1Data(in := fbRotaryTable.ActualPosition + OneStep) THEN
				IF Buffer_Station4.Add1Data(in := fbRotaryTable.ActualPosition + 2*OneStep) THEN
					TableRegister := 20;

				END_IF				
			END_IF
		END_IF
END_CASE


(* Table sequences *)
CASE RotaryTableProcess OF
	0://Idle
		IF Buffer_RotaryTable.Count > 0 THEN
			RotaryTableProcess := 10;
		END_IF
	10:
		fbRotaryTable.MR_MoveRelative(lrRelativeDistance := Buffer_RotaryTable.GetValue);
		IF NOT fbRotaryTable.Busy THEN
//			iRTCVision.M_CommandStation1(); // change to station 3
//			IF NOT iRTCVision.Busy THEN
//				;
//			END_IF
			;
		END_IF
END_CASE
///}}}
END_METHOD

METHOD MR_Start : BOOL
(* 
Button START on the HMI
*)
fbMsgAutoStarted.Send(0);

IF eMachineStateAuto = MACHINE_STATE_AUTO_IDLE THEN
	eMachineState := MACHINE_STATE_AUTO;
	eMachineStateAuto := MACHINE_STATE_AUTO_RUNNING;
	bStop := FALSE;
	
END_IF

MR_Start := TRUE;
END_METHOD

METHOD MR_Stop : BOOL
VAR_INPUT
END_VAR
bRunning := FALSE;

IF eMachineStateAuto = MACHINE_STATE_AUTO_RUNNING THEN
	eMachineStateAuto := MACHINE_STATE_AUTO_IDLE;
	
END_IF
END_METHOD

METHOD PROTECTED MS_Aborting
(* 
Add here code to abort all machine objects's e.g robots, axes, cylinders. 
At the end add "eMachineState := MACHINE_STATE_UNINITIALIZED;" to finish aborting.
*)
CASE eMachineStateAbort OF
	MACHINE_STATE_ABORTING_TABLE:
		fbRotaryTable.MR_Abort();
		IF NOT fbRotaryTable.Active THEN
			eMachineState := MACHINE_STATE_UNINITIALIZED;
		eMachineStateUninitialized := MACHINE_STATE_UNINITIALIZED_DONE;
		END_IF
		
	MACHINE_STATE_ABORTING_ROBOT_CYCLE_STOP:
		IF fbRobot.ref_CR800.ErrorOccuring THEN			
			eMachineStateAbort := MACHINE_STATE_ABORTING_TABLE;
			eMachineState := MACHINE_STATE_UNINITIALIZED;
			eMachineStateUninitialized := MACHINE_STATE_UNINITIALIZED_DONE;
		ELSE
			fbRobot.ref_CR800.MR_CycleStop();
			IF NOT fbRobot.ref_CR800.Busy THEN
				eMachineStateAbort := MACHINE_STATE_ABORTING_TABLE;
				eMachineState := MACHINE_STATE_UNINITIALIZED;
				eMachineStateUninitialized := MACHINE_STATE_UNINITIALIZED_DONE;
			END_IF
		END_IF

END_CASE
END_METHOD

METHOD PROTECTED MS_Auto
VAR_INST
	bSetSP:BOOL;
	rSp:REAL;
END_VAR
CASE eMachineStateAuto OF
	MACHINE_STATE_AUTO_IDLE:
		bRunning := FALSE;
		
	MACHINE_STATE_AUTO_RUNNING:
		bRunning := TRUE;
		//Test();
		Production_fixing();
		//Robot_Process();
		//TableProcess();
		//tableRefer();
		//robotcamtest();
		//Robot_Process();
		
END_CASE

(*========== HMI control =============*)
(* Bowl feeder *)
IF btnStartBowl THEN
	fbBowlFeeder.MR_Start();
	doBlowBowlFeeder.Out := TRUE;
END_IF

IF btnStopBowl THEN
	fbBowlFeeder.MR_Stop();
	doBlowBowlFeeder.Out := FALSE;
END_IF

fbBowlFeeder.Setpoint := rBowlFeederSetpoint;
END_METHOD

METHOD PROTECTED MS_AutoToManual
VAR_INPUT
END_VAR
(* 
Add here code to switch machine into manual mode. 
At the end add "eMachineState := MACHINE_STATE_MANUAL;" to finish switching.
*)
(* Switching mode to manual simulation - DELETE *)
//tonTestDelay(IN := TRUE, PT:= T#500MS);
//bRunning := FALSE;
//IF tonTestDelay.Q THEN
//	tonTestDelay(IN := FALSE);
//	eMachineState := MACHINE_STATE_MANUAL;
//END_IF

bRunning := FALSE;
eMachineState := MACHINE_STATE_MANUAL;
END_METHOD

METHOD PROTECTED MS_Emergency
VAR_INPUT
END_VAR
END_METHOD

METHOD PROTECTED MS_Initializing
VAR_INST
	uBowlFeederInitState : UINT;
	uTableInitState : UINT;
	uVisionInitState : UINT;
	
END_VAR
(* 
Add here code to initialize all machine objects's e.g robots, axes, cylinders. 
At the end add "eMachineState := MACHINE_STATE_READY_INITIALIZED;" to finish initialization.
*)
CASE eMachineStateInit OF
	MACHINE_STATE_INITIALIZING_MACHINE_LOGGER:
		fbMachineLogger.MR_Init();
		IF NOT fbMachineLogger.Busy THEN
			eMachineStateInit := MACHINE_STATE_INITIALIZING_ROBOT_CONTROLERS_RESET;
		END_IF
(*	
	MACHINE_STATE_INITIALIZING_RECIPES_MANAGER:
		IF stShell.stPlatform.ref_fbRecipesManager.Active THEN
			eMachineStateInit := MACHINE_STATE_INITIALIZING_CLEAR_ALL_ERRORS;
		END_IF
		
	MACHINE_STATE_INITIALIZING_CLEAR_ALL_ERRORS:
		stShell.stPlatform.ref_fbAlarmControler.MR_ClearAll(TRUE);
		IF NOT stShell.stPlatform.ref_fbAlarmControler.Busy THEN
			//eMachineStateInit := MACHINE_STATE_INITIALIZING_MES_COMMAND_LOGGER;
			eMachineStateInit := MACHINE_STATE_INITIALIZING_SAFETY_INITIALIZATION;
		END_IF
	
	MACHINE_STATE_INITIALIZING_SAFETY_INITIALIZATION:
		stShell.stPlatform.ref_MachineSafety.RunStop := TRUE;
		tonDelay( IN := TRUE, PT := T#3S);
		IF tonDelay.Q THEN
			tonDelay(IN := FALSE);
			//fbMessageSafetySystemRestarted.Send(0); (* TC_Alarm *)
			eMachineStateInit := MACHINE_STATE_INITIALIZING_CHECK_ESTOP;
		END_IF
	
	MACHINE_STATE_INITIALIZING_CHECK_ESTOP:
		poDoorLock.Out := FALSE;
		IF stShell.stPlatform.ref_MachineSafety.E_Stop AND stShell.stPlatform.ref_MachineSafety.ExternalE_Stop THEN
			eMachineStateInit := MACHINE_STATE_INITIALIZING_CHECK_DOOR_LOCKS;
		END_IF
	
	MACHINE_STATE_INITIALIZING_CHECK_DOOR_LOCKS:
		IF NOT stShell.stPlatform.ref_MachineSafety.E_Stop OR NOT stShell.stPlatform.ref_MachineSafety.ExternalE_Stop THEN
			eMachineStateInit := MACHINE_STATE_INITIALIZING_CHECK_ESTOP;		
		ELSE
			IF stShell.stPlatform.ref_MachineSafety.SafetyOverride THEN
				eMachineStateInit := MACHINE_STATE_INITIALIZING_ROBOTS_POWER_CHECK;
			ELSE
				poDoorLock.Out := TRUE;
				IF stShell.stPlatform.ref_MachineSafety.DoorLock THEN
					eMachineStateInit := MACHINE_STATE_INITIALIZING_ROBOTS_POWER_CHECK;
				END_IF
			END_IF
		END_IF
	
	MACHINE_STATE_INITIALIZING_ROBOTS_POWER_CHECK:
		IF fbRobot.ref_CR800.CR800PoweredOn THEN
			eMachineStateInit := MACHINE_STATE_INITIALIZING_SAFETY_RESET;
		END_IF
	
	MACHINE_STATE_INITIALIZING_SAFETY_RESET:
		stShell.stPlatform.ref_MachineSafety.ErrorAck := TRUE;
		eMachineStateInit := MACHINE_STATE_INITIALIZING_SAFETY_START;
	
	MACHINE_STATE_INITIALIZING_SAFETY_START:
		stShell.stPlatform.ref_MachineSafety.ErrorAck := FALSE;
		IF NOT stShell.stPlatform.ref_MachineSafety.E_Stop OR NOT stShell.stPlatform.ref_MachineSafety.ExternalE_Stop THEN
			eMachineStateInit := MACHINE_STATE_INITIALIZING_CHECK_ESTOP;		
		ELSIF NOT stShell.stPlatform.ref_MachineSafety.SafetyOverride AND NOT stShell.stPlatform.ref_MachineSafety.DoorLock THEN
			eMachineStateInit := MACHINE_STATE_INITIALIZING_CHECK_DOOR_LOCKS;
		ELSE
			poResetButtonLight.Out := TRUE;
			IF stShell.stPlatform.ref_MachineSafety.RestartButton THEN
				poResetButtonLight.Out := FALSE;
				eMachineStateInit := MACHINE_STATE_INITIALIZING_ROBOT_CONTROLERS_RESET;
			END_IF
		END_IF
	*)
	MACHINE_STATE_INITIALIZING_ROBOT_CONTROLERS_RESET:
		fbRobot.ref_CR800.MR_Reset();
		IF NOT fbRobot.ref_CR800.Busy THEN
			uTableInitState := 10;
			uBowlFeederInitState := 10;
			eMachineStateInit := MACHINE_STATE_INITIALIZING_ROBOT_AUTO_MODE_SW;
		END_IF
(*
	MACHINE_STATE_INITIALIZING_SAFETY_CHECK:
		IF NOT stShell.stPlatform.ref_MachineSafety.FB_Error AND NOT stShell.stPlatform.ref_MachineSafety.FB_Error THEN
			fbRobot.ModeSwitch := TRUE;
			eMachineStateInit := MACHINE_STATE_INITIALIZING_ROBOT_ABORT;
		END_IF
	*)
	
	MACHINE_STATE_INITIALIZING_ROBOT_AUTO_MODE_SW:
		fbRobot.ModeSwitch := TRUE;
		eMachineStateInit := MACHINE_STATE_INITIALIZING_ROBOT_ABORT;
		
	MACHINE_STATE_INITIALIZING_ROBOT_ABORT:
		fbRobot.MR_Abort();
		IF NOT fbRobot.Active THEN
			eMachineStateInit := MACHINE_STATE_INITIALIZING_ROBOT_INIT;
		END_IF
	
	MACHINE_STATE_INITIALIZING_ROBOT_INIT:
		fbRobot.MR_Init();
		IF fbRobot.Active THEN
			eMachineStateInit := MACHINE_STATE_INITIALIZING_ROBOT_HOME;
		END_IF
	
	MACHINE_STATE_INITIALIZING_ROBOT_HOME:
		fbRobot.MR_GoHome();
		IF NOT fbRobot.Busy THEN
			eMachineStateInit := MACHINE_STATE_INITIALIZING_ROBOT_AUTOMATIC_MODE;
		END_IF
	
	MACHINE_STATE_INITIALIZING_ROBOT_AUTOMATIC_MODE:
		fbRobot.ref_CR800.MR_GoAuto();
		IF NOT fbRobot.ref_CR800.Busy THEN
			eMachineStateInit := MACHINE_STATE_INITIALIZING_DONE;
		END_IF
	
//	MACHINE_STATE_INITIALIZING_ROTARY_TABLE_ABORT:
		

//	MACHINE_STATE_INITIALIZING_ROTARY_TABLE_INIT:
		

//	MACHINE_STATE_INITIALIZING_ROTARY_TABLE_HOME:
		
		
//	MACHINE_STATE_INITIALIZING_BOWL_INIT:
		

	MACHINE_STATE_INITIALIZING_DONE:
		IF uTableInitState = 30 AND uBowlFeederInitState = 20 THEN	(* check Table and bowl init done *)
			eMachineStateInit := MACHINE_STATE_INITIALIZING_MACHINE_LOGGER;
			eMachineState := MACHINE_STATE_READY_INITIALIZED;
		END_IF
		
END_CASE
/////////////////////////////////////////////////////////
CASE uTableInitState OF
	0://idle
		;
	5:
		fbRotaryTable.MR_Abort();
		IF NOT fbRotaryTable.PowerOn THEN
			uTableInitState := 10;
		END_IF
	10://init
		fbRotaryTable.MR_Init();
		IF fbRotaryTable.PowerOn THEN
			uTableInitState := 20;
		END_IF
	20://homing
		fbRotaryTable.MR_Home(lrHomePosition := DEFAULT_HOME_POSITION );
		IF fbRotaryTable.IsHomed THEN
			uTableInitState := 30;
		END_IF
	30://done
		;
END_CASE
/////////////////////////////////////////////////////////
CASE uBowlFeederInitState OF
	0://idle
		;
	10:
		fbBowlFeeder.MR_Init();
		IF NOT fbBowlFeeder.Busy THEN
			uBowlFeederInitState := 20;
		END_IF
	20://done
		;
END_CASE
END_METHOD

METHOD PROTECTED MS_Manual
VAR_INPUT
END_VAR
(* 
Leave empty - manual mode is provided by HMI controler and automatic frame generator.
*)
;
END_METHOD

METHOD PROTECTED MS_ManualToAuto
VAR_INPUT
END_VAR
(* 
Add here code to switch machine into auto mode. 
At the end add "eMachineState := MACHINE_STATE_AUTO;" to finish switching.
*)
//CASE eMachineStateManualToAuto OF
//	MACHINE_STATE_MANUAL_TO_AUTO_ROBOT_CYCLE_STOP:
//		IF arrRobot[0].ErrorOccuring THEN
//			eMachineStateManualToAuto := MACHINE_STATE_MANUAL_TO_AUTO_ROBOT_ABORT;
//		ELSE
//			arrRobot[0].MR_CycleStop();
//			IF NOT arrRobot[0].Busy THEN
//				eMachineStateManualToAuto := MACHINE_STATE_MANUAL_TO_AUTO_ROBOT_ABORT;
//			END_IF
//		END_IF
		
//	MACHINE_STATE_MANUAL_TO_AUTO_ROBOT_ABORT:
//		arrRobot[0].MR_Abort();
//		IF NOT arrRobot[0].Active THEN
//			//eMachineStateManualToAuto := MACHINE_STATE_MANUAL_TO_AUTO_ROBOT_REMOTE_MODE;
//			eMachineStateManualToAuto := MACHINE_STATE_MANUAL_TO_AUTO_ROBOT_INIT;
//		END_IF
	
////	MACHINE_STATE_MANUAL_TO_AUTO_ROBOT_REMOTE_MODE:
////		poRobotModeSwitch.Out := TRUE;
////		tonDelay( IN := TRUE, PT:= T#500MS);
////		IF tonDelay.Q THEN
////			tonDelay(IN := FALSE);
////			eMachineStateManualToAuto := MACHINE_STATE_MANUAL_TO_AUTO_ROBOT_ONE_INIT;
////		END_IF
		
//	MACHINE_STATE_MANUAL_TO_AUTO_ROBOT_INIT:
//		arrRobot[0].MR_Init();
//		IF arrRobot[0].Active THEN
//			eMachineStateManualToAuto := MACHINE_STATE_MANUAL_TO_AUTO_ROBOT_HOME;
//		END_IF
		
//	MACHINE_STATE_MANUAL_TO_AUTO_ROBOT_HOME:
//		arrRobot[0].MR_GoHome();
//		IF NOT arrRobot[0].Busy THEN
//			eMachineStateManualToAuto := MACHINE_STATE_MANUAL_TO_AUTO_ROBOT_AUTOMATIC_MODE;
//		END_IF
		
//	MACHINE_STATE_MANUAL_TO_AUTO_ROBOT_AUTOMATIC_MODE:
//		arrRobot[0].MR_GoAuto();
//		IF NOT arrRobot[0].Busy THEN
//			eMachineStateManualToAuto := MACHINE_STATE_MANUAL_TO_AUTO_DONE;
//		END_IF
		
//	MACHINE_STATE_MANUAL_TO_AUTO_DONE:
//		eMachineStateManualToAuto := MACHINE_STATE_MANUAL_TO_AUTO_ROBOT_CYCLE_STOP;
//		eMachineState := MACHINE_STATE_AUTO;
		
//END_CASE
END_METHOD

METHOD PROTECTED MS_ReadyInitialized
VAR_INPUT
END_VAR
(*
Add code here if some internal parameters are needed to set after initialization or leave it default.
At the end add "eMachineState := MACHINE_STATE_AUTO;" to finish and go to IDLE state.
*)
eMachineStateInit := MACHINE_STATE_INITIALIZING_MACHINE_LOGGER;
eMachineState := MACHINE_STATE_AUTO;
eMachineStateAuto := MACHINE_STATE_AUTO_IDLE;
eMachineStateAutoAOI := MACHINE_STATE_AUTO_AOI_IDLE;
END_METHOD

METHOD PROTECTED MS_Reset
VAR_INPUT
END_VAR
(* 
Add here code to reset all machine objects's e.g robots, axes, cylinders. 
At the end add "eMachineState := MACHINE_STATE_RESET_DONE;" to finish reseting.
*)
(* Reset simulation - DELETE  *)
//tonTestDelay(IN := TRUE, PT:= T#4S);
//IF tonTestDelay.Q THEN
//	tonTestDelay(IN := FALSE);
//	eMachineState := MACHINE_STATE_RESET_DONE;
//END_IF

eMachineState := MACHINE_STATE_RESET_DONE;
END_METHOD

METHOD PROTECTED MS_ResetDone
VAR_INPUT
END_VAR
eMachineState := eMachineStateBeforeReset;
END_METHOD

METHOD PROTECTED MS_Uninitialized

VAR_INST
	btestmethodcam: BOOL;
	btestasd : bool;
END_VAR
VAR
	
END_VAR
CASE eMachineStateUninitialized OF
	
	MACHINE_STATE_UNINITIALIZED_POWER_ON_CR800:
		IF fbRobot.ref_CR800.CR800PoweredOn THEN
			eMachineStateUninitialized := MACHINE_STATE_UNINITIALIZED_CR800_ETHERCAT_STATUS_CHECK;
		END_IF
	
	MACHINE_STATE_UNINITIALIZED_CR800_ETHERCAT_STATUS_CHECK:
		IF fbRobot.M_EtherCATStatusCheck() THEN
			eMachineStateUninitialized := MACHINE_STATE_UNINITIALIZED_DONE;
		END_IF

	MACHINE_STATE_UNINITIALIZED_DONE:
		eMachineStateInit := MACHINE_STATE_INITIALIZING_MACHINE_LOGGER;
	
END_CASE
END_METHOD

METHOD PROTECTED Production : BOOL
VAR_INST
	(* Robot *)
	RobotState 					: UINT;
	
	(* Table *)
	TableState					: UINT;
	OneStep 					: LREAL:= -60.0; //-61.1928;	(* Define by the distance between station 3 and 4 *)
	lrRelativeDistance 			: LREAL;
	bProductAboveTable 			: BOOL;				(* Signal Robot is at the table *)
	bGetPictureStation3			: BOOL; 			(* Cmd get picture st3 to vision system *)
	bGetPictureStation4 		: BOOL; 			(* Cmd get picture st4 to vision system *)
	bResultProcessing 			: BOOL;				(* Request result from vision system, then add buffer for sorting station *)
	
	(* Buffer *)
	BufferState : UINT;
	Buffer_RotaryTable			: FB_DataSetFifo_1; 	(* Contain the position of all product on the table *)
	Buffer_Station3				: FB_DataSetFifo_1;	(* Contain the trigger position *)
	Buffer_Station4				: FB_DataSetFifo_1;	(* Contain the trigger position *)
	
	(* Sorting Station *)
	Buffer_SortGood				: FB_DataSetFifo_1;
	Buffer_SortDirt				: FB_DataSetFifo_1;
	Buffer_SortDent				: FB_DataSetFifo_1;
	Buffer_SortReject			: FB_DataSetFifo_1;
	
	
	
	lrSortGoodPos				: LREAL;
	lrSortDirtPos				: LREAL;
	lrSortDentPos				: LREAL;
	lrSortRejectPos				: LREAL;
	
	uSortGoodGetPosState		: UINT; 			(* state machine of get sort position from buffer *)
	uSortDirtGetPosState		: UINT;
	uSortDentGetPosState		: UINT;
	uSortRejectGetPosState		: UINT;
		
	tonGoodDelay				: TON;				(* one shoot of good delay valve *)
	tonDirtDelay				: TON;				(* one shoot of dirt delay valve *)
	tonDentDelay				: TON;				(* one shoot of dent delay valve *)								
	tonRejectDelay				: TON;				(* one shoot of reject delay valve *)	
							

	
	(*=== Vision ===*)
	Vision3State 		: UINT;
	Vision4State		: UINT;
	lrCapPosStation3 	: LREAL;
	lrCapPosStation4	: LREAL;
	bGood 				: BOOL;
	bAtVision3 			: BOOL;	(* Product is at vision 3 *)
	bAtVision4 			: BOOL;	(* Product is at vision 4 *)
	eFinalResult		: E_VisionResult;

	(* Axis status flags *)
	bActive					: BOOL;
	bBusy					: BOOL;								(* Function block currently executes one of the requests *)
	bError					: BOOL;								(* Error status flag *)
	iErrorID				: UDINT;							(* Error ID *)
	iAxisErrorID			: UDINT;							(* Axis error ID*)
	lrActualPosition		: LREAL;							(* Actual axis position in selected units *)
	rActualVelocity			: REAL;								(* Actual axis velocity in selected units *)
	bPowerOn 				: BOOL;								(* Power On status bit *)
	bIsHomed				: BOOL;								(* Axis has been homed even once *)
	bInVelocity				: BOOL;								(* Axis is moving in target velocity *)
	bInPostion				: BOOL;								(* Axis reached target position *)
	bMoveActive				: BOOL;								(* Axis is moving to target position *)
	bJogDone				: BOOL;								(* Axis manual movement by jog done *)
	bStopped				: BOOL;								(* Axis movement has been stopped *)
	bHalted					: BOOL;								(* Axis movement has been halted *)
	eStatePlcOpen			: E_AxisStatePlcOpen;
	
	uBufferTableCount : UDINT;
	
	(* testing bit *)
	bResultTest : BOOL;
	bResultGood : BOOL;
	bResultDirt : BOOL;
	bResultDent : BOOL;
	bResultReject : BOOL;

END_VAR
///(*==================================== Robot + Vision process ====================================*){{{
CASE RobotState OF	
	0://IDLE go bowl
		fbRobot.MR_GoBowl();
		IF NOT fbRobot.Busy THEN
			RobotState := 5;
		END_IF		
	5://product detected
		IF diProductPresenceBowl.In THEN (* waiting product *)
			RobotState := 6;
		END_IF
	
	6://go input
		fbRobot.MR_GoInputProduct();
		IF NOT fbRobot.Busy THEN
			RobotState := 7;
		END_IF
		
	7://robot pick
		fbRobot.MR_Pick();
		IF NOT fbRobot.Busy THEN
			RobotState := 10;
		END_IF 
		
	10://go to station 1
		fbRobot.MR_GoStation1();
		IF NOT fbRobot.Busy THEN
			RobotState := 20;
		END_IF
		
	20://double trig cam 1+2
		IF doTriggerCam1.Command(PulseWidth:=T#1MS, DelayTimeForSecondTrigger := T#35MS) AND
			doTriggerCam2.Command(PulseWidth:=T#1MS, DelayTimeForSecondTrigger := T#35MS) THEN
			RobotState:= 30;
		END_IF
	30://go to station 2
		fbRobot.MR_GoStation2();
		IF NOT fbRobot.Busy THEN
			RobotState := 40;
		END_IF
	40://double trig cam 3+4
		IF doTriggerCam3.Command(PulseWidth:=T#1MS, DelayTimeForSecondTrigger := T#35MS) AND
			doTriggerCam4.Command(PulseWidth:=T#1MS, DelayTimeForSecondTrigger := T#35MS) THEN
			RobotState := 50;
		END_IF
	50://goto rotary table
		fbRobot.MR_GoRotaryTable();
		IF NOT fbRobot.Busy THEN
			bProductAboveTable := TRUE;		
			RobotState:= 60;
		END_IF
	60://waiting command from table
		;
		
END_CASE
///============================================================================================}}}
///(*==================================== Table process ====================================*){{{
CASE TableState OF
	0:// idle | waiting for product
		IF bProductAboveTable THEN
			TableState:= 10;
		END_IF
	10://command place product and reset robot sequence
		fbRobot.MR_Place();
		IF NOT fbRobot.Busy THEN
			bProductAboveTable := FALSE;
			RobotState := 0;
			TableState := 20;
		END_IF
	20://add buffer for st 3+4, table
		Buffer_RotaryTable.A_Add(in:= OneStep);
		Buffer_RotaryTable.A_Add(in:= OneStep);
		Buffer_Station3.A_Add(in:= fbRotaryTable.ActualPosition + OneStep);
		Buffer_Station4.A_Add(in:= fbRotaryTable.ActualPosition + 2*OneStep);
		TableState := 30;
		
//	21://get vision 3capture position
//		IF Vision3State = 0 THEN
//			Vision3State:= 10;
//			TableState:=22;
//		END_IF
//	22://get vision 4 capture position
//		IF Vision4State = 0 THEN
//			Vision4State:= 10;
//			TableState:=30;
//		END_IF
	
	30://get table distance movement
		Buffer_RotaryTable.A_Remove(out => lrRelativeDistance);
		TableState := 40;
	40://move distance
		fbRotaryTable.MR_MoveRelative(lrRelativeDistance);
		IF fbRotaryTable.InPosition THEN
			
			TableState := 41;
		END_IF
		
	41:// check position of vision station 3
		IF Vision3State = 0 THEN
			TableState := 42;
		END_IF
	42:
		Buffer_Station3.A_Get(out => lrCapPosStation3);
		bGetPictureStation3 := TRUE;
		
		IF LREAL_TO_INT(fbRotaryTable.ActualPosition) = LREAL_TO_INT(lrCapPosStation3) THEN
			Buffer_Station3.A_Remove(out => lrCapPosStation3);
			Vision3State:= 30;
			TableState := 43;
			
		ELSE
			bGetPictureStation3 := FALSE;
			TableState := 43;
			
		END_IF
			
	43:// check position of vision station 4
		IF Vision4State = 0 THEN
			TableState := 44;
		END_IF
	44:
		Buffer_Station4.A_Get(out => lrCapPosStation4);
		bGetPictureStation4 := TRUE;
		bResultProcessing := TRUE;
		
		IF LREAL_TO_INT(fbRotaryTable.ActualPosition) = LREAL_TO_INT(lrCapPosStation4) THEN
			Buffer_Station4.A_Remove(out => lrCapPosStation4);
			Vision4State:= 30;
			TableState := 60;
			
		ELSE
			bGetPictureStation4 := FALSE;
			bResultProcessing := FALSE;
			TableState := 60;
			
		END_IF
	
	
	
	
//	50://command vision 3
//		IF Vision3State = 0 THEN
//			Vision3State:= 20;
//			TableState:=55;
//		END_IF
//	55:	//command vision 4
//		IF Vision4State = 0 THEN
//			Vision4State:= 20;
//			TableState:=60;
//		END_IF

	
	
	
	
	60://check taking picture done
		IF NOT bGetPictureStation3 AND NOT bGetPictureStation4  AND NOT bResultProcessing THEN
			TableState := 70;
		END_IF
		
	70://state check result | product above table | buffer | go through sorting station
		IF bProductAboveTable THEN
			TableState := 10;//take product
		ELSIF Buffer_RotaryTable.nCount > 0 THEN
			TableState := 30;//get distance
		ELSE
			(* Make sure that the product is sorted *)
			fbRotaryTable.MR_MoveRelative(2*OneStep);
			IF fbRotaryTable.InPosition THEN
				
				TableState := 0;
			END_IF
			
		END_IF
	
END_CASE
///============================================================================================}}}
///(*==================================== Vision 3+4 process ====================================*){{{
CASE Vision3State OF
	0://idle | waiting
		;
//	10://get position in buffer
//		Buffer_Station3.A_Remove(out => lrCapPosStation3);
//		Vision3State := 0;

//	20://check position with table
//		bGetPictureStation3 := TRUE;
//		IF LREAL_TO_INT(fbRotaryTable.ActualPosition) = LREAL_TO_INT(lrCapPosStation3) THEN //convert from lreal to int for less precise
//			Vision3State:= 30;
//		ELSE
//			bGetPictureStation3 := FALSE;
//			Vision3State:= 0;
//		END_IF
			
	30://take picture cam 5+6
		IF doTriggerCam5.Command(PulseWidth:= T#1MS, DelayTimeForSecondTrigger:= T#34MS) AND
			doTriggerCam6.Command(PulseWidth:= T#1MS, DelayTimeForSecondTrigger:= T#34MS) THEN
			
			bGetPictureStation3 := FALSE;
			Vision3State := 0; 
		END_IF
		
END_CASE

(* station 4 have to take picture and request result from system *)
CASE Vision4State OF
	0:
		;
//	10://get trigger position in buffer
//		Buffer_Station4.A_Remove(out => lrCapPosStation4);
//		Vision4State := 0;

//	20://check trigger position with table position
//		bGetPictureStation4 := TRUE;
//		bResultProcessing 	:= TRUE;
//		IF LREAL_TO_INT(fbRotaryTable.ActualPosition) = LREAL_TO_INT(lrCapPosStation4) THEN //convert from lreal to int for less precise
//			Vision4State:= 30;
//		ELSE
//			bResultProcessing			:= FALSE;
//			bGetPictureStation4 		:= FALSE;
//			Vision4State:= 0;
//		END_IF
	
	30://trigger cam 7
		IF doTriggerCam7.Command(PulseWidth:= T#1MS, DelayTimeForSecondTrigger:= T#33MS) THEN
			bGetPictureStation4 := FALSE;
			Vision4State:= 40;
		END_IF
		
	40://request result
		(* testing purpose *)
		bResultGood:= TRUE;
		IF bResultGood THEN
			eFinalResult := VISION_RESULT_GOOD;
			bResultGood := FALSE;
			Vision4State:= 0;
		ELSIF bResultDirt THEN
			eFinalResult := VISION_RESULT_CONTAMINATION_DIRTY;
			bResultDirt := FALSE;
			Vision4State:= 0;
		ELSIF bResultDent THEN
			eFinalResult := VISION_RESULT_SCRATCH_DENT;
			bResultDent := FALSE;
			Vision4State:= 0;
		ELSIF bResultReject THEN
			eFinalResult := VISION_RESULT_REJECT;
			bResultReject := FALSE;
			Vision4State:= 0;
		END_IF

